# B&R Automation Studio project TD52 (part 62)

```c
  /* End of Outputs for SubSystem: '<S306>/2nd Order Filter1' */

  /* Outputs for Atomic SubSystem: '<S306>/2nd Order Filter2' */
  Gen2_ref_undOrderFilter(rtb_p2HP,
    Gen2_ref_B->BusInput3.fdc.r2ndOrdFiltOmegaPressure,
    Gen2_ref_B->BusInput3.fdc.r2ndOrdFiltDPressure, rtb_bResetBdc,
    &Gen2_ref_B->undOrderFilter2, &Gen2_ref_DWork->undOrderFilter2, inst);

  /* End of Outputs for SubSystem: '<S306>/2nd Order Filter2' */

  /* Outputs for Atomic SubSystem: '<S306>/2nd Order Filter3' */
  Gen2_ref_undOrderFilter3(rtb_p2s,
    Gen2_ref_B->BusInput3.fdc.r2ndOrdFiltOmegaPressure,
    Gen2_ref_B->BusInput3.fdc.r2ndOrdFiltDPressure, rtb_bResetBdc,
    &Gen2_ref_B->undOrderFilter3, &Gen2_ref_DWork->undOrderFilter3, inst);

  /* End of Outputs for SubSystem: '<S306>/2nd Order Filter3' */

  /* Switch: '<S272>/Switch2' */
  if (Gen2_ref_B->BusInput3.fdc.bEnable2ndOrdFiltDerivative) {
    /* Switch: '<S272>/Switch6' incorporates:
     *  Constant: '<S307>/Constant2'
     *  DiscreteIntegrator: '<S307>/Discrete-Time Integrator'
     *  Product: '<S307>/Product'
     *  Product: '<S307>/Product1'
     *  Sum: '<S307>/Sum'
     *  Sum: '<S307>/Sum4'
     */
    if (Gen2_ref_B->BusInput3.fdc.bEnableTransSwFilt) {
      rtb_Switch2_gd_idx_0 = (1.0 -
        Gen2_ref_DWork->DiscreteTimeIntegrator_DSTATE_d) *
        Gen2_ref_B->sf_FILTERnodelay.d_dt +
        Gen2_ref_DWork->DiscreteTimeIntegrator_DSTATE_d *
        Gen2_ref_B->undOrderFilter.Switch1;
      rtb_Switch2_gd_idx_1 = (1.0 -
        Gen2_ref_DWork->DiscreteTimeIntegrator_DSTATE_d) *
        Gen2_ref_B->sf_FILTERnodelay1.d_dt +
        Gen2_ref_DWork->DiscreteTimeIntegrator_DSTATE_d *
        Gen2_ref_B->undOrderFilter1.Switch1;
      rtb_Switch2_gd_idx_2 = (1.0 -
        Gen2_ref_DWork->DiscreteTimeIntegrator_DSTATE_d) *
        Gen2_ref_B->sf_FILTERnodelay2.d_dt +
        Gen2_ref_DWork->DiscreteTimeIntegrator_DSTATE_d *
        Gen2_ref_B->undOrderFilter2.Switch1;
      rtb_Switch2_gd_idx_3 = (1.0 -
        Gen2_ref_DWork->DiscreteTimeIntegrator_DSTATE_d) *
        Gen2_ref_B->sf_FILTERnodelay3.d_dt +
        Gen2_ref_DWork->DiscreteTimeIntegrator_DSTATE_d *
        Gen2_ref_B->undOrderFilter3.Switch1;
    } else {
      rtb_Switch2_gd_idx_0 = Gen2_ref_B->undOrderFilter.Switch1;
      rtb_Switch2_gd_idx_1 = Gen2_ref_B->undOrderFilter1.Switch1;
      rtb_Switch2_gd_idx_2 = Gen2_ref_B->undOrderFilter2.Switch1;
      rtb_Switch2_gd_idx_3 = Gen2_ref_B->undOrderFilter3.Switch1;
    }

    /* End of Switch: '<S272>/Switch6' */
  } else {
    rtb_Switch2_gd_idx_0 = Gen2_ref_B->sf_FILTERnodelay.d_dt;
    rtb_Switch2_gd_idx_1 = Gen2_ref_B->sf_FILTERnodelay1.d_dt;
    rtb_Switch2_gd_idx_2 = Gen2_ref_B->sf_FILTERnodelay2.d_dt;
    rtb_Switch2_gd_idx_3 = Gen2_ref_B->sf_FILTERnodelay3.d_dt;
  }

  /* End of Switch: '<S272>/Switch2' */

  /* DataTypeConversion: '<S4>/Data Type Conversion1' */
  rtb_Product1_b = Gen2_ref_B->BusInput.tT.rT1LP;

  /* Outputs for Atomic SubSystem: '<S196>/T1LP_filt' */
  /* Bias: '<S4>/C2K' */
  Gen2_ref_N_TC_HP_filt(rtb_Product1_b + 273.15,
                        Gen2_ref_B->BusInput3.inFilt.rTiF_T, rtb_bResetBdc,
                        &Gen2_ref_B->T1LP_filt, &Gen2_ref_DWork->T1LP_filt, inst);

  /* End of Outputs for SubSystem: '<S196>/T1LP_filt' */

  /* DataTypeConversion: '<S4>/Data Type Conversion8' */
  rtb_Product1_b = Gen2_ref_B->BusInput.tT.rT1HP;

  /* Outputs for Atomic SubSystem: '<S195>/T1HP_filt' */
  /* Bias: '<S4>/C2K1' */
  Gen2_ref_N_TC_HP_filt(rtb_Product1_b + 273.15,
                        Gen2_ref_B->BusInput3.inFilt.rTiF_T, rtb_bResetBdc,
                        &Gen2_ref_B->T1HP_filt, &Gen2_ref_DWork->T1HP_filt, inst);

  /* End of Outputs for SubSystem: '<S195>/T1HP_filt' */

  /* Outputs for Atomic SubSystem: '<S267>/Mg' */
  Gen2_ref_Mg(Gen2_ref_B->BusInput3.eng.rRho_gas, &Gen2_ref_B->Mg, inst);

  /* End of Outputs for SubSystem: '<S267>/Mg' */

  /* Sum: '<S342>/Sum2' */
  rtb_Switch1_k = u0;

  /* Abs: '<S342>/Abs3' */
  rtb_Switch_jv = fabs(rtb_Switch1_k);

  /* Sum: '<S381>/Add1' */
  rtb_Product1_b = Gen2_ref_B->BusInput3.EGTLim.rT_CR_soft -
    Gen2_ref_B->BusInput3.EGTLim.rT_CR_hard;

  /* Saturate: '<S381>/Saturation6' */
  if (rtb_Product1_b > 1.0E+6) {
    rtb_Saturation6 = 1.0E+6;
  } else if (rtb_Product1_b < 1.0) {
    rtb_Saturation6 = 1.0;
  } else {
    rtb_Saturation6 = rtb_Product1_b;
  }

  /* End of Saturate: '<S381>/Saturation6' */

  /* DataTypeConversion: '<S4>/Data Type Conversion12' */
  rtb_Product1_b = Gen2_ref_B->BusInput.tT.rTcylMax;

  /* Bias: '<S342>/Bias' incorporates:
   *  Bias: '<S4>/C2K5'
   */
  rtb_PactOut_o = (rtb_Product1_b + 273.15) + -273.15;

  /* Sum: '<S381>/Add6' */
  rtb_Divide6_n = Gen2_ref_B->BusInput3.EGTLim.rT_max -
    Gen2_ref_B->BusInput3.EGTLim.rT_CR_hard;

  /* Sum: '<S381>/Sum15' */
  rtb_Switch2_n5 = (rtb_PactOut_o + rtb_Saturation6) - rtb_Divide6_n;

  /* Switch: '<S387>/Switch2' incorporates:
   *  Constant: '<S381>/Constant17'
   *  RelationalOperator: '<S387>/LowerRelop1'
   *  RelationalOperator: '<S387>/UpperRelop'
   *  Switch: '<S387>/Switch'
   */
  if (rtb_Switch2_n5 > rtb_Saturation6) {
    rtb_Switch2_n5 = rtb_Saturation6;
  } else if (rtb_Switch2_n5 < 0.0) {
    /* Switch: '<S387>/Switch' incorporates:
     *  Constant: '<S381>/Constant17'
     */
    rtb_Switch2_n5 = 0.0;
  }

  /* End of Switch: '<S387>/Switch2' */

  /* Switch: '<S381>/Switch7' incorporates:
   *  Constant: '<S381>/Constant23'
   *  Constant: '<S381>/Constant5'
   *  Product: '<S381>/Divide8'
   *  Sum: '<S381>/Sum1'
   */
  if (Gen2_ref_B->BusInput3.EGTLim.bActive) {
    rtb_Product1_b = 1.0 - rtb_Switch2_n5 / rtb_Saturation6;
  } else {
    rtb_Product1_b = 1.0;
  }

  /* End of Switch: '<S381>/Switch7' */

  /* Product: '<S342>/Product' */
  rtb_Product1_b *= rtb_Switch_jv;

  /* Switch: '<S380>/Switch2' incorporates:
   *  RelationalOperator: '<S380>/LowerRelop1'
   */
  if (!(rtb_Switch1_k > rtb_Product1_b)) {
    /* Gain: '<S342>/Gain2' */
    rtb_Switch_jv = -rtb_Switch_jv;

    /* Switch: '<S380>/Switch' incorporates:
     *  RelationalOperator: '<S380>/UpperRelop'
     */
    if (rtb_Switch1_k < rtb_Switch_jv) {
      rtb_Product1_b = rtb_Switch_jv;
    } else {
      rtb_Product1_b = rtb_Switch1_k;
    }

    /* End of Switch: '<S380>/Switch' */
  }

  /* End of Switch: '<S380>/Switch2' */

  /* Gain: '<S342>/Gain4' */
  rtb_Switch_jv = -1.0E-6 * rtb_Product1_b;

  /* Sum: '<S11>/Sum' incorporates:
   *  Constant: '<S11>/Constant'
   */
  rtb_Switch_fy_tmp_tmp = 1.0 - Gen2_ref_B->BusInput.IN_EC_rGT_RatioMix_TC2;
  rtb_Product1_b = 1.0 - Gen2_ref_B->BusInput.IN_EC_rGT_RatioMix_TC2;

  /* Saturate: '<S11>/Saturation' */
  if (rtb_Product1_b > 1.0) {
    rtb_Product1_b = 1.0;
  } else if (rtb_Product1_b < 0.0) {
    rtb_Product1_b = 0.0;
  }

  /* End of Saturate: '<S11>/Saturation' */

  /* Saturate: '<S11>/Saturation1' */
  if (Gen2_ref_B->BusInput.IN_EC_rGT_RatioMix_TC2 > 1.0F) {
    rtb_rPos_CBV3 = 1.0F;
  } else if (Gen2_ref_B->BusInput.IN_EC_rGT_RatioMix_TC2 < 0.0F) {
    rtb_rPos_CBV3 = 0.0F;
  } else {
    rtb_rPos_CBV3 = Gen2_ref_B->BusInput.IN_EC_rGT_RatioMix_TC2;
  }

  /* End of Saturate: '<S11>/Saturation1' */

  /* Sum: '<S11>/Sum1' incorporates:
   *  Product: '<S11>/Product'
   *  Product: '<S11>/Product1'
   */
  rtb_Sum1_idx_2 = rtb_Product1_b * Gen2_ref_B->BusInput3.eng.rMin_Air_Ratio_kg
    + rtb_rPos_CBV3 * Gen2_ref_B->BusInput3.eng.rMin_Air_Ratio_M_kg;
  rtb_Sum1_idx_3 = rtb_Product1_b * Gen2_ref_B->BusInput3.eng.rLHV +
    rtb_rPos_CBV3 * Gen2_ref_B->BusInput3.eng.rLHV_M;

  /* Switch: '<S3>/etaVolConst' */
  if (Gen2_ref_B->BusInput3.Eff.bActive_EtaVolExt) {
    rtb_etaVolConst_lt = Gen2_ref_B->BusInput3.Eff.rEtaVolExt;
  } else {
    rtb_etaVolConst_lt = 0.0;
  }

  /* End of Switch: '<S3>/etaVolConst' */

  /* Switch: '<S3>/etaBreakConst' */
  if (Gen2_ref_B->BusInput3.Eff.bActive_EtaBrakeExt) {
    rtb_etaBreakConst = Gen2_ref_B->BusInput3.Eff.rEtaBrakeExt;
  } else {
    rtb_etaBreakConst = 0.0;
  }

  /* End of Switch: '<S3>/etaBreakConst' */

  /* Switch: '<S342>/Switch' */
  if (Gen2_ref_B->BusInput3.PowCtrl.bActive_MbcFF) {
    /* Product: '<S340>/Divide1' incorporates:
     *  Constant: '<S340>/Constant'
     *  Constant: '<S340>/R_air'
     */
    rtb_Switch1_k = rtb_Sum1_idx_2 * 287.15 * Gen2_ref_B->T2s_filt.Switch *
      rtb_kW2W1_h * 12.566370614359172;

    /* Saturate: '<S340>/Saturation1' */
    if (rtb_Switch1_k <= 1.0) {
      rtb_Switch1_k = 1.0;
    }

    /* End of Saturate: '<S340>/Saturation1' */

    /* Saturate: '<S340>/Saturation' */
    if (rtb_Sum1_idx_2 <= 1.0) {
      rtb_Product1_b = 1.0;
    } else {
      rtb_Product1_b = rtb_Sum1_idx_2;
    }

    /* End of Saturate: '<S340>/Saturation' */

    /* Sum: '<S340>/Sum' incorporates:
     *  Constant: '<S340>/Constant1'
     *  Gain: '<S340>/Gain'
     *  Product: '<S340>/Divide'
     *  Product: '<S340>/Divide2'
     *  Product: '<S340>/Divide4'
     */
    rtb_Switch_e3 = Gen2_ref_B->BusInput3.eng.rVol_Hub_Eng * rtb_Sum1_idx_3 *
      (0.10471975511965977 * Gen2_ref_B->BusInput3.eng.rN_Nom) *
      rtb_etaVolConst_lt * rtb_etaBreakConst * Gen2_ref_B->p2s_filt.Switch /
      rtb_Switch1_k - 1.0 / rtb_Product1_b;

    /* Saturate: '<S340>/Saturation2' */
    if (rtb_Switch_e3 > 2.2) {
      rtb_Switch_e3 = 2.2;
    } else if (rtb_Switch_e3 < 1.3) {
      rtb_Switch_e3 = 1.3;
    }

    /* End of Saturate: '<S340>/Saturation2' */
  } else {
    rtb_Switch_e3 = Gen2_ref_B->BusInput3.PowCtrl.rLam_ff;
  }

  /* End of Switch: '<S342>/Switch' */

  /* Switch: '<S381>/Switch8' incorporates:
   *  Constant: '<S381>/Constant10'
   *  Product: '<S381>/Product'
   *  Product: '<S381>/Product1'
   *  Sum: '<S381>/Sum16'
   */
  if (Gen2_ref_B->BusInput3.EGTLim.bActive) {
    /* Sum: '<S381>/Sum8' */
    u0 = rtb_PactOut_o - rtb_Divide6_n;

    /* Saturate: '<S381>/Saturation3' */
    if (u0 > 1.0E+6) {
      u0 = 1.0E+6;
    } else if (u0 < 0.0) {
      u0 = 0.0;
    }

    /* End of Saturate: '<S381>/Saturation3' */
    rtb_Switch8 = u0 * Gen2_ref_B->BusInput3.EGTLim.rKaw_hard +
      Gen2_ref_B->BusInput3.EGTLim.rKaw_soft * rtb_Switch2_n5;
  } else {
    rtb_Switch8 = 0.0;
  }

  /* End of Switch: '<S381>/Switch8' */

  /* Gain: '<S14>/Gain2' incorporates:
   *  Gain: '<S133>/Gain1'
   *  Gain: '<S14>/Gain'
   *  Gain: '<S14>/Gain3'
   *  Gain: '<S23>/Gain'
   *  Gain: '<S25>/Gain1'
   *  Gain: '<S426>/Gain1'
   *  Gain: '<S9>/Gain5'
   *  Switch: '<S106>/Switch2'
   *  Switch: '<S133>/Switch'
   *  Switch: '<S133>/Switch1'
   *  Switch: '<S426>/Switch'
   *  Switch: '<S426>/Switch1'
   *  Switch: '<S426>/Switch2'
   *  Switch: '<S494>/etaVolConst'
   */
  rtb_kW2W1_h = 1.0E-5 * Gen2_ref_B->p2s_filt.Switch;
  rtb_Product1_b = rtb_kW2W1_h;

  /* S-Function (sfix_look1_dyn): '<S14>/Lookup Table Dynamic1' */
  /* Dynamic Look-Up Table Block: '<S14>/Lookup Table Dynamic1'
   * Input0  Data Type:  Floating Point real_T
   * Input1  Data Type:  Floating Point real_T
   * Input2  Data Type:  Floating Point real_T
   * Output0 Data Type:  Floating Point real_T
   * Saturation Mode: Saturate
   * Lookup Method: Linear_Endpoint
   *
   */
  LookUp_real_T_real_T_SAT( &(rtb_Sum8_m),
    &Gen2_ref_B->BusInput3.LamLim.refPoint_LamUpLim_ABS_y[0], rtb_Product1_b,
    &Gen2_ref_B->BusInput3.LamLim.refPoint_LamUpLim_ABS_x[0], 5U, inst);

  /* Logic: '<S14>/Logical Operator6' incorporates:
   *  Logic: '<S14>/Logical Operator10'
   */
  rtb_LogicalOperator5_g_tmp =
    !Gen2_ref_B->BusInput3.LamLim.bActLamLim_GQCimprovement;

  /* Logic: '<S14>/Logical Operator5' incorporates:
   *  Logic: '<S14>/Logical Operator6'
   */
  rtb_LogicalOperator5_mv = (Gen2_ref_B->BusInput3.LamLim.bLamOffsInitPerm ||
    rtb_LogicalOperator5_g_tmp);

  /* Gain: '<S14>/Gain3' */
  rtb_Product1_b = rtb_kW2W1_h;

  /* S-Function (sfix_look1_dyn): '<S14>/Lookup Table Dynamic2' */
  /* Dynamic Look-Up Table Block: '<S14>/Lookup Table Dynamic2'
   * Input0  Data Type:  Floating Point real_T
   * Input1  Data Type:  Floating Point real_T
   * Input2  Data Type:  Floating Point real_T
   * Output0 Data Type:  Floating Point real_T
   * Saturation Mode: Saturate
   * Lookup Method: Linear_Endpoint
   *
   */
  LookUp_real_T_real_T_SAT( &(rtb_LookupTableDynamic2),
    &Gen2_ref_B->BusInput3.LamLim.refPoint_LamLoLim_ABS_y[0], rtb_Product1_b,
    &Gen2_ref_B->BusInput3.LamLim.refPoint_LamLoLim_ABS_x[0], 5U, inst);

  /* Saturate: '<S14>/Saturation' */
  if (Gen2_ref_B->BusInput3.LamLim.rFactEnrich <= 0.0) {
    rtb_Product1_b = 0.0;
  } else {
    rtb_Product1_b = Gen2_ref_B->BusInput3.LamLim.rFactEnrich;
  }

  /* End of Saturate: '<S14>/Saturation' */

  /* Gain: '<S14>/Gain' */
  rtb_PactOut_o = rtb_kW2W1_h;

  /* Switch: '<S14>/Switch5' */
  if (Gen2_ref_B->BusInput3.LamLim.bNOx250mg) {
    /* S-Function (sfix_look1_dyn): '<S14>/Lookup Table Dynamic' */
    /* Dynamic Look-Up Table Block: '<S14>/Lookup Table Dynamic'
     * Input0  Data Type:  Floating Point real_T
     * Input1  Data Type:  Floating Point real_T
     * Input2  Data Type:  Floating Point real32_T
     * Output0 Data Type:  Floating Point real_T
     * Saturation Mode: Saturate
     * Lookup Method: Linear_Endpoint
     *
     */
    LookUp_real_Treal32_T_K4km1JJi( &(rtb_LookupTableDynamic_n),
      &Gen2_ref_B->BusInput3.LamLim.rLamMapBase250mg[0], rtb_PactOut_o,
      &Gen2_ref_B->BusInput3.LamLim.rPr_p2s_Lup_in[0], 9U, inst);
    rtb_PactOut_o = rtb_LookupTableDynamic_n;
  } else {
    /* S-Function (sfix_look1_dyn): '<S14>/Lookup Table Dynamic3' */
    /* Dynamic Look-Up Table Block: '<S14>/Lookup Table Dynamic3'
     * Input0  Data Type:  Floating Point real_T
     * Input1  Data Type:  Floating Point real_T
     * Input2  Data Type:  Floating Point real32_T
     * Output0 Data Type:  Floating Point real_T
     * Saturation Mode: Saturate
     * Lookup Method: Linear_Endpoint
     *
     */
    LookUp_real_Treal32_T_K4km1JJi( &(rtb_LookupTableDynamic3),
      &Gen2_ref_B->BusInput3.LamLim.rLamMapBase[0], rtb_PactOut_o,
      &Gen2_ref_B->BusInput3.LamLim.rPr_p2s_Lup_in[0], 9U, inst);
    rtb_PactOut_o = rtb_LookupTableDynamic3;
  }

  /* End of Switch: '<S14>/Switch5' */

  /* Product: '<S14>/Product' incorporates:
   *  Constant: '<S14>/Constant'
   *  Sum: '<S14>/Sum1'
   *  Sum: '<S14>/Sum2'
   */
  rtb_Product_l0 = (1.0 - rtb_Product1_b) * (rtb_PactOut_o -
    rtb_LookupTableDynamic2);

  /* Delay: '<S14>/Resettable Delay2' */
  if (Gen2_ref_DWork->icLoad_l) {
    Gen2_ref_DWork->ResettableDelay2_DSTATE =
      Gen2_ref_B->BusInput3.LamLim.rLamOffsetLimInit;
  }

  rtb_Product1_b = Gen2_ref_DWork->ResettableDelay2_DSTATE;

  /* End of Delay: '<S14>/Resettable Delay2' */

  /* Switch: '<S14>/Switch6' incorporates:
   *  DataTypeConversion: '<S4>/Data Type Conversion28'
   *  DataTypeConversion: '<S4>/Data Type Conversion31'
   *  DataTypeConversion: '<S4>/Data Type Conversion32'
   *  Sum: '<S14>/Sum16'
   *  UnitDelay: '<S14>/Unit Delay4'
   */
  if (Gen2_ref_DWork->UnitDelay4_DSTATE_d) {
    rtb_Divide6_n = (((Gen2_ref_B->BusInput.rLam_idle - rtb_LookupTableDynamic2)
                      - rtb_Product_l0) - Gen2_ref_B->BusInput.rOffsetLamLimit)
      + Gen2_ref_B->BusInput.rDeltaLamSync;
  } else {
    rtb_Divide6_n = rtb_Product1_b;
  }

  /* End of Switch: '<S14>/Switch6' */

  /* Switch: '<S14>/Switch7' */
  if (rtb_LogicalOperator5_mv) {
    rtb_Switch2_n5 = Gen2_ref_B->BusInput3.LamLim.rLamOffsetLimInit;
  } else {
    rtb_Switch2_n5 = rtb_Divide6_n;
  }

  /* End of Switch: '<S14>/Switch7' */

  /* Delay: '<S14>/Resettable Delay' incorporates:
   *  Logic: '<Root>/Logical Operator'
   */
  Gen2_ref_DWork->icLoad_i =
    ((((Gen2_ref_PrevZCSigState->ResettableDelay_Reset_ZCE_j == 1) != (int32_T)
       rtb_LogicalOperator_cn) &&
      (Gen2_ref_PrevZCSigState->ResettableDelay_Reset_ZCE_j != 3)) ||
     rtb_LogicalOperator_cn || Gen2_ref_DWork->icLoad_i);
  Gen2_ref_PrevZCSigState->ResettableDelay_Reset_ZCE_j = rtb_LogicalOperator_cn;
  if (Gen2_ref_DWork->icLoad_i) {
    Gen2_ref_DWork->ResettableDelay_DSTATE_l = rtb_Switch2_n5;
  }

  /* Sum: '<S14>/Sum' incorporates:
   *  DataTypeConversion: '<S4>/Data Type Conversion28'
   *  UnitDelay: '<S14>/Unit Delay'
   */
  rtb_Switch1_k = (Gen2_ref_DWork->UnitDelay_DSTATE -
                   Gen2_ref_B->BusInput.rOffsetLamLimit) - rtb_PactOut_o;

  /* Switch: '<S14>/Switch9' */
  if (rtb_Switch2_jv) {
    /* Switch: '<S860>/Switch2' incorporates:
     *  Constant: '<S14>/Constant2'
     *  Delay: '<S14>/Resettable Delay'
     *  RelationalOperator: '<S860>/LowerRelop1'
     *  RelationalOperator: '<S860>/UpperRelop'
     *  Switch: '<S860>/Switch'
     */
    if (rtb_Switch1_k > 2.0) {
      rtb_Switch1_k = 2.0;
    } else if (rtb_Switch1_k < Gen2_ref_DWork->ResettableDelay_DSTATE_l) {
      /* Switch: '<S860>/Switch' incorporates:
       *  Delay: '<S14>/Resettable Delay'
       */
      rtb_Switch1_k = Gen2_ref_DWork->ResettableDelay_DSTATE_l;
    }

    /* End of Switch: '<S860>/Switch2' */
  }

  /* End of Switch: '<S14>/Switch9' */

  /* Abs: '<S858>/Abs' */
  rtb_Product1_b = rtb_Product1_e_tmp;

  /* Switch: '<S858>/Switch' incorporates:
   *  Constant: '<S858>/Constant2'
   *  RelationalOperator: '<S858>/Relational Operator'
   */
  if (2.2204460492503131E-16 >= rtb_Product1_b) {
    rtb_bResetHlci_0 = 2.2204460492503131E-16;
  } else {
    rtb_bResetHlci_0 = Gen2_ref_B->BusInput3.eng.rP_Nom;
  }

  /* End of Switch: '<S858>/Switch' */

  /* RelationalOperator: '<S14>/Relational Operator' incorporates:
   *  Gain: '<S14>/Gain1'
   *  Product: '<S14>/Divide'
   */
  rtb_RelationalOperator_l5 = (0.001 * rtb_Gain2_ao / rtb_bResetHlci_0 >
    Gen2_ref_B->BusInput3.LamLim.rPminSSadapt);

  /* Switch: '<S908>/Switch' incorporates:
   *  Constant: '<S908>/Constant2'
   *  RelationalOperator: '<S908>/Relational Operator'
   */
  if (2.2204460492503131E-16 >= rtb_Product1_b) {
    rtb_bResetHlci_0 = 2.2204460492503131E-16;
  } else {
    rtb_bResetHlci_0 = Gen2_ref_B->BusInput3.eng.rP_Nom;
  }

  /* End of Switch: '<S908>/Switch' */

  /* Product: '<S20>/Divide1' incorporates:
   *  Gain: '<S20>/Gain6'
   */
  rtb_Saturation6 = 0.001 * rtb_Gain2_ao / rtb_bResetHlci_0;

  /* Outputs for Atomic SubSystem: '<S20>/Filter1' */
  /* Logic: '<Root>/Logical Operator' */
  Gen2_ref_Filter3(rtb_Saturation6, Gen2_ref_B->BusInput3.LamLim.rTiSSfilter,
                   Gen2_ref_ConstB.T_filt1, rtb_LogicalOperator_cn,
                   &Gen2_ref_B->Filter1_ny, &Gen2_ref_DWork->Filter1_ny, inst);

  /* End of Outputs for SubSystem: '<S20>/Filter1' */

  /* Logic: '<S917>/Logical Operator' incorporates:
   *  Logic: '<Root>/Logical Operator'
   *  UnitDelay: '<S917>/Unit Delay'
   */
  rtb_LogicalOperator_i = (rtb_LogicalOperator_cn ||
    Gen2_ref_DWork->UnitDelay_DSTATE_k);

  /* DiscreteIntegrator: '<S917>/Discrete-Time Integrator' */
  if (rtb_LogicalOperator_i || (Gen2_ref_DWork->DiscreteTimeIntegrator_PrevR_ka
       != 0)) {
    Gen2_ref_DWork->DiscreteTimeIntegrator_DSTATE_c = 0.0;
  }

  /* RelationalOperator: '<S917>/Relational Operator' incorporates:
   *  DiscreteIntegrator: '<S917>/Discrete-Time Integrator'
   */
  rtb_RelationalOperator_a = (Gen2_ref_B->BusInput3.LamLim.rTiSSsampling <=
    Gen2_ref_DWork->DiscreteTimeIntegrator_DSTATE_c);

  /* Outputs for Enabled SubSystem: '<S20>/Enabled Subsystem2' incorporates:
   *  EnablePort: '<S909>/Enable'
   */
  if (rtb_RelationalOperator_a) {
    /* Inport: '<S909>/In1' */
    Gen2_ref_B->In1 = Gen2_ref_B->Filter1_ny.Switch;

    /* Memory: '<S909>/Memory' */
    FILT_IN = Gen2_ref_DWork->Memory_PreviousInput;

    /* Sum: '<S909>/Sum' */
    Gen2_ref_B->Sum = Gen2_ref_B->In1 - FILT_IN;

    /* Update for Memory: '<S909>/Memory' */
    Gen2_ref_DWork->Memory_PreviousInput = Gen2_ref_B->In1;
  }

  /* End of Outputs for SubSystem: '<S20>/Enabled Subsystem2' */

  /* Sum: '<S20>/Sum2' */
  rtb_Product1_b = rtb_Saturation6 - Gen2_ref_B->In1;

  /* Abs: '<S20>/Abs4' */
  rtb_Saturation6 = fabs(rtb_Product1_b);

  /* Outputs for Atomic SubSystem: '<S20>/Filter3' */
  /* Logic: '<Root>/Logical Operator' */
  Gen2_ref_Filter3(rtb_Saturation6, Gen2_ref_B->BusInput3.LamLim.rTiSSfilter,
                   Gen2_ref_ConstB.T_filt1, rtb_LogicalOperator_cn,
                   &Gen2_ref_B->Filter3_f, &Gen2_ref_DWork->Filter3_f, inst);

  /* End of Outputs for SubSystem: '<S20>/Filter3' */

  /* Abs: '<S20>/Abs1' */
  rtb_Product1_b = fabs(Gen2_ref_B->Sum);

  /* RelationalOperator: '<S20>/Relational Operator3' */
  rtb_LogicalOperator_aw = (rtb_Product1_b <=
    Gen2_ref_B->BusInput3.LamLim.rThrshSSPow);

  /* Gain: '<S20>/Gain1' incorporates:
   *  Sum: '<S20>/Sum'
   */
  rtb_Product1_b = (Gen2_ref_B->p2s_filt.Switch - rtb_Divide_kt) * 0.01;

  /* Abs: '<S20>/Abs' */
  rtb_Abs = fabs(rtb_Product1_b);

  /* Gain: '<S20>/Gain2' */
  rtb_Product1_b = 2.0 * Gen2_ref_B->BusInput3.LamLim.rThrshSSboost;

  /* Outputs for Atomic SubSystem: '<S20>/Filter' */
  /* Logic: '<Root>/Logical Operator' */
  Gen2_ref_Filter3(rtb_Abs, Gen2_ref_B->BusInput3.LamLim.rTiSSfilter,
                   Gen2_ref_ConstB.T_filt1, rtb_LogicalOperator_cn,
                   &Gen2_ref_B->Filter_f, &Gen2_ref_DWork->Filter_f, inst);

  /* End of Outputs for SubSystem: '<S20>/Filter' */

  /* Outputs for Atomic SubSystem: '<S20>/TON1' */
  /* Logic: '<S20>/Logical Operator' incorporates:
   *  RelationalOperator: '<S20>/Relational Operator'
   *  RelationalOperator: '<S20>/Relational Operator1'
   */
  Gen2_ref_TON_1(((rtb_Abs <= rtb_Product1_b) && (Gen2_ref_B->Filter_f.Switch <=
    Gen2_ref_B->BusInput3.LamLim.rThrshSSboost)),
                 Gen2_ref_B->BusInput3.LamLim.rTiSSsampling, &Gen2_ref_B->TON1_n,
                 &Gen2_ref_DWork->TON1_n, inst);

  /* End of Outputs for SubSystem: '<S20>/TON1' */

  /* Sum: '<S20>/Sum1' incorporates:
   *  DataTypeConversion: '<S4>/Data Type Conversion16'
   */
  rtb_Product1_b = rtb_DataTypeConversion15 - Gen2_ref_B->BusInput.rN_Set;

  /* Abs: '<S20>/Abs3' */
  rtb_Abs = fabs(rtb_Product1_b);

  /* Gain: '<S20>/Gain3' */
  rtb_Product1_b = 2.0 * Gen2_ref_B->BusInput3.LamLim.rThrshSSspeed;

  /* Outputs for Atomic SubSystem: '<S20>/Filter2' */
  /* Logic: '<Root>/Logical Operator' */
  Gen2_ref_Filter3(rtb_Abs, Gen2_ref_B->BusInput3.LamLim.rTiSSfilter,
                   Gen2_ref_ConstB.T_filt1, rtb_LogicalOperator_cn,
                   &Gen2_ref_B->Filter2_o, &Gen2_ref_DWork->Filter2_o, inst);

  /* End of Outputs for SubSystem: '<S20>/Filter2' */

  /* Outputs for Atomic SubSystem: '<S20>/TON' */
  /* Logic: '<S20>/Logical Operator2' incorporates:
   *  RelationalOperator: '<S20>/Relational Operator4'
   *  RelationalOperator: '<S20>/Relational Operator5'
   */
  Gen2_ref_TON_1(((rtb_Abs <= rtb_Product1_b) && (Gen2_ref_B->Filter2_o.Switch <=
    Gen2_ref_B->BusInput3.LamLim.rThrshSSspeed)),
                 Gen2_ref_B->BusInput3.LamLim.rTiSSsampling, &Gen2_ref_B->TON_l,
                 &Gen2_ref_DWork->TON_l, inst);

  /* End of Outputs for SubSystem: '<S20>/TON' */

  /* Outputs for Atomic SubSystem: '<S20>/TON2' */
  /* Logic: '<S20>/Logical Operator1' incorporates:
   *  RelationalOperator: '<S20>/Relational Operator2'
   *  RelationalOperator: '<S20>/Relational Operator6'
   */
  Gen2_ref_TON_1(((rtb_Saturation6 <= Gen2_ref_B->BusInput3.LamLim.rThrshSSPow) &&
                  (Gen2_ref_B->Filter3_f.Switch <=
                   Gen2_ref_B->BusInput3.LamLim.rThrshSSPow) &&
                  rtb_LogicalOperator_aw && Gen2_ref_B->TON1_n.LogicalOperator3 &&
                  Gen2_ref_B->TON_l.LogicalOperator3),
                 Gen2_ref_B->BusInput3.LamLim.rTiSSsampling, &Gen2_ref_B->TON2,
                 &Gen2_ref_DWork->TON2, inst);

  /* End of Outputs for SubSystem: '<S20>/TON2' */

  /* Switch: '<S14>/Switch4' incorporates:
   *  Delay: '<S14>/Resettable Delay'
   *  Logic: '<S14>/Logical Operator1'
   *  Switch: '<S14>/Switch3'
   */
  if (rtb_RelationalOperator_l5 &&
      Gen2_ref_B->BusInput3.LamLim.bAutomaticOffsetON &&
      (Gen2_ref_B->BusInput3.LamLim.bActLambdaOffsetNotSteady ||
       Gen2_ref_B->TON2.LogicalOperator3)) {
    /* Switch: '<S14>/Switch12' */
    if (rtb_Switch4_mu) {
      /* Switch: '<S861>/Switch2' incorporates:
       *  Constant: '<S14>/Constant6'
       *  Delay: '<S14>/Resettable Delay'
       *  RelationalOperator: '<S861>/LowerRelop1'
       *  RelationalOperator: '<S861>/UpperRelop'
       *  Switch: '<S861>/Switch'
       */
      if (rtb_Switch1_k > Gen2_ref_DWork->ResettableDelay_DSTATE_l) {
        rtb_Switch1_k = Gen2_ref_DWork->ResettableDelay_DSTATE_l;
      } else if (rtb_Switch1_k < -2.0) {
        /* Switch: '<S861>/Switch' incorporates:
         *  Constant: '<S14>/Constant6'
         */
        rtb_Switch1_k = -2.0;
      }

      /* End of Switch: '<S861>/Switch2' */
    }

    /* End of Switch: '<S14>/Switch12' */
  } else {
    rtb_Switch1_k = Gen2_ref_DWork->ResettableDelay_DSTATE_l;
  }

  /* End of Switch: '<S14>/Switch4' */

  /* Switch: '<S14>/Switch10' incorporates:
   *  Logic: '<S14>/Logical Operator7'
   *  Logic: '<S14>/Logical Operator9'
   *  Product: '<S14>/Divide1'
   */
  if (Gen2_ref_B->TON2.LogicalOperator3 ||
      (!Gen2_ref_B->BusInput3.LamLim.bActLambdaOffsetNotSteady)) {
    rtb_bResetHlci_0 = Gen2_ref_B->BusInput3.LamLim.rTiFiltLambdaOffset;
  } else {
    rtb_bResetHlci_0 = Gen2_ref_B->BusInput3.LamLim.rFactTiFiltLamOffsNotSteady *
      Gen2_ref_B->BusInput3.LamLim.rTiFiltLambdaOffset;
  }

  /* End of Switch: '<S14>/Switch10' */

  /* Outputs for Atomic SubSystem: '<S14>/Filter' */
  /* Logic: '<Root>/Logical Operator' */
  Gen2_ref_Pd_filt(rtb_Switch1_k, rtb_bResetHlci_0, rtb_Switch2_n5,
                   rtb_LogicalOperator_cn, &Gen2_ref_B->Filter_l,
                   &Gen2_ref_DWork->Filter_l, inst);

  /* End of Outputs for SubSystem: '<S14>/Filter' */

  /* Sum: '<S14>/Sum4' incorporates:
   *  DataTypeConversion: '<S4>/Data Type Conversion28'
   */
  rtb_Sum4_ny = Gen2_ref_B->Filter_l.Switch +
    Gen2_ref_B->BusInput.rOffsetLamLimit;

  /* Saturate: '<S14>/Saturation1' */
  if (Gen2_ref_B->BusInput3.LamLim.rFactLean <= 0.0) {
    rtb_Product1_b = 0.0;
  } else {
    rtb_Product1_b = Gen2_ref_B->BusInput3.LamLim.rFactLean;
  }

  /* End of Saturate: '<S14>/Saturation1' */

  /* Product: '<S14>/Product1' incorporates:
   *  Constant: '<S14>/Constant1'
   *  Sum: '<S14>/Sum6'
   *  Sum: '<S14>/Sum7'
   */
  rtb_Product1_b = (rtb_PactOut_o - rtb_Sum8_m) * (1.0 - rtb_Product1_b);

  /* Sum: '<S14>/Sum5' */
  rtb_Sum5_j = rtb_Sum4_ny + rtb_Product1_b;

  /* Sum: '<S14>/Sum3' */
  rtb_Switch2_n5 = rtb_Sum8_m + rtb_Sum5_j;

  /* MinMax: '<S14>/MinMax' */
  if ((!(rtb_Switch2_n5 <= Gen2_ref_B->BusInput3.LamLim.rLam_max)) && (!rtIsNaN
       (Gen2_ref_B->BusInput3.LamLim.rLam_max))) {
    rtb_Switch2_n5 = Gen2_ref_B->BusInput3.LamLim.rLam_max;
  }

  /* End of MinMax: '<S14>/MinMax' */

  /* Sum: '<S14>/Sum8' */
  rtb_Sum8_m = rtb_Sum4_ny + rtb_Product_l0;

  /* Delay: '<S14>/Resettable Delay3' incorporates:
   *  Logic: '<Root>/Logical Operator'
   */
  Gen2_ref_DWork->icLoad_f =
    ((((Gen2_ref_PrevZCSigState->ResettableDelay3_Reset_ZCE == 1) != (int32_T)
       rtb_LogicalOperator_cn) &&
      (Gen2_ref_PrevZCSigState->ResettableDelay3_Reset_ZCE != 3)) ||
     rtb_LogicalOperator_cn || Gen2_ref_DWork->icLoad_f);
  Gen2_ref_PrevZCSigState->ResettableDelay3_Reset_ZCE = rtb_LogicalOperator_cn;
  Gen2_ref_DWork->ResettableDelay3_DSTATE = (Gen2_ref_DWork->icLoad_f ||
    Gen2_ref_DWork->ResettableDelay3_DSTATE);

  /* Switch: '<S14>/Switch13' incorporates:
   *  Constant: '<S14>/Constant5'
   *  Delay: '<S14>/Resettable Delay3'
   *  Logic: '<S14>/Logical Operator11'
   */
  if (Gen2_ref_DWork->ResettableDelay3_DSTATE) {
    rtb_RelationalOperator_l5 = !rtb_RelationalOperator_l5;
  } else {
    rtb_RelationalOperator_l5 = false;
  }

  /* End of Switch: '<S14>/Switch13' */

  /* Logic: '<S14>/Logical Operator12' */
  rtb_LogicalOperator12_a = !rtb_RelationalOperator_l5;

  /* Switch: '<S14>/Switch11' incorporates:
   *  Logic: '<Root>/Logical Operator'
   *  Logic: '<S14>/Logical Operator4'
   */
  if (rtb_LogicalOperator_cn || rtb_LogicalOperator12_a ||
      rtb_LogicalOperator5_g_tmp) {
    /* Sum: '<S14>/Sum9' */
    rtb_Switch1_k = rtb_LookupTableDynamic2 + rtb_Sum8_m;

    /* MinMax: '<S14>/MinMax1' */
    if ((!(rtb_Switch1_k >= Gen2_ref_B->BusInput3.LamLim.rLam_min)) && (!rtIsNaN
         (Gen2_ref_B->BusInput3.LamLim.rLam_min))) {
      rtb_Switch1_k = Gen2_ref_B->BusInput3.LamLim.rLam_min;
    }
  } else {
    /* Sum: '<S14>/Sum9' */
    u0 = rtb_LookupTableDynamic2 + rtb_Sum8_m;

    /* MinMax: '<S14>/MinMax1' */
    if ((!(u0 >= Gen2_ref_B->BusInput3.LamLim.rLam_min)) && (!rtIsNaN
         (Gen2_ref_B->BusInput3.LamLim.rLam_min))) {
      u0 = Gen2_ref_B->BusInput3.LamLim.rLam_min;
    }

    /* Sum: '<S14>/Sum14' incorporates:
     *  DataTypeConversion: '<S4>/Data Type Conversion31'
     *  DataTypeConversion: '<S4>/Data Type Conversion32'
     */
    rtb_Switch1_k = (real_T)Gen2_ref_B->BusInput.rLam_idle +
      Gen2_ref_B->BusInput.rDeltaLamSync;

    /* MinMax: '<S14>/MinMax4' */
    if ((u0 >= rtb_Switch1_k) || rtIsNaN(rtb_Switch1_k)) {
      rtb_Switch1_k = u0;
    }

    /* End of MinMax: '<S14>/MinMax4' */
  }

  /* End of Switch: '<S14>/Switch11' */

  /* Outputs for Atomic SubSystem: '<S342>/PID_Power' */
  /* Product: '<S379>/Divide1' */
  FILT_IN = Gen2_ref_B->BusInput3.PowCtrl.rKp * rtb_Switch_jv;

  /* BusCreator: '<Root>/Bus Creator' incorporates:
   *  BusCreator: '<S379>/Bus Creator1'
   *  DataTypeConversion: '<S379>/Data Type Conversion1'
   *  Outport: '<Root>/dbg'
   */
  Gen2_ref_Y->dbg.HLC.BGen2DbgHlcPowCtrl.up = (real32_T)FILT_IN;

  /* Product: '<S379>/Divide2' */
  r = rtb_Switch_jv * Gen2_ref_B->BusInput3.PowCtrl.rKd;

  /* DiscreteIntegrator: '<S379>/Discrete-Time Integrator1' */
  if (rtb_LogicalOperator_in || (Gen2_ref_DWork->DiscreteTimeIntegrator1_PrevR_l
       != 0)) {
    Gen2_ref_DWork->DiscreteTimeIntegrator1_DSTA_nh = 0.0;
  }

  /* Product: '<S379>/Divide3' incorporates:
   *  DiscreteIntegrator: '<S379>/Discrete-Time Integrator1'
   *  Sum: '<S379>/Sum1'
   */
  rtb_Divide3_p = (r - Gen2_ref_DWork->DiscreteTimeIntegrator1_DSTA_nh) *
    Gen2_ref_B->BusInput3.PowCtrl.rN;

  /* Delay: '<S379>/Delay2' */
  r = Gen2_ref_DWork->Delay2_DSTATE_o;

  /* MATLAB Function: '<S379>/MATLAB Function' incorporates:
   *  Constant: '<S342>/Constant'
   *  Sum: '<S379>/Sum6'
   */
  Gen2_ref_MATLABFunction_g(rtb_LogicalOperator_in, 0.0, rtb_LogicalOperator1_e,
    ((r - rtb_Switch_e3) - FILT_IN) - rtb_Divide3_p,
    &Gen2_ref_B->sf_MATLABFunction_g, &Gen2_ref_DWork->sf_MATLABFunction_g, inst);

  /* DiscreteIntegrator: '<S379>/Discrete-Time Integrator' */
  if (Gen2_ref_DWork->DiscreteTimeIntegrator_IC_LOA_g != 0) {
    Gen2_ref_DWork->DiscreteTimeIntegrator_DSTATE_f =
      Gen2_ref_B->sf_MATLABFunction_g.Y0Out;
  }

  if (Gen2_ref_B->sf_MATLABFunction_g.ireset ||
      (Gen2_ref_DWork->DiscreteTimeIntegrator_PrevR_o3 != 0)) {
    Gen2_ref_DWork->DiscreteTimeIntegrator_DSTATE_f =
      Gen2_ref_B->sf_MATLABFunction_g.Y0Out;
  }

  /* Sum: '<S379>/Sum3' incorporates:
   *  DiscreteIntegrator: '<S379>/Discrete-Time Integrator'
   *  Sum: '<S379>/Sum'
   */
  FILT_IN = ((FILT_IN + Gen2_ref_DWork->DiscreteTimeIntegrator_DSTATE_f) +
             rtb_Divide3_p) + rtb_Switch_e3;

  /* Product: '<S385>/delta rise limit' incorporates:
   *  SampleTimeMath: '<S385>/sample time'
   *
   * About '<S385>/sample time':
   *  y = K where K = ( w * Ts )
   */
  r = Gen2_ref_B->BusInput3.PowCtrl.rLam_Sr_Pos * 0.01;

  /* Delay: '<S385>/Delay' incorporates:
   *  Delay: '<S404>/Delay'
   */
  Gen2_ref_DWork->icLoad_nq = ((((Gen2_ref_PrevZCSigState->Delay_Reset_ZCE_at ==
    1) != (int32_T)rtb_LogicalOperator_in) &&
    (Gen2_ref_PrevZCSigState->Delay_Reset_ZCE_at != 3)) ||
    rtb_LogicalOperator_in || Gen2_ref_DWork->icLoad_nq);
  Gen2_ref_PrevZCSigState->Delay_Reset_ZCE_at = rtb_LogicalOperator_in;
  if (Gen2_ref_DWork->icLoad_nq) {
    Gen2_ref_DWork->Delay_DSTATE_dj = rtb_Switch_e3;
  }

  /* Switch: '<S385>/etaVolConst' */
  if (rtb_LogicalOperator_in) {
    rtb_Abs = rtb_Switch_e3;
  } else {
    rtb_Abs = FILT_IN;
  }

  /* End of Switch: '<S385>/etaVolConst' */

  /* Sum: '<S385>/Difference Inputs1' incorporates:
   *  Delay: '<S385>/Delay'
   */
  rtb_Saturation6 = rtb_Abs - Gen2_ref_DWork->Delay_DSTATE_dj;

  /* Switch: '<S386>/Switch2' incorporates:
   *  RelationalOperator: '<S386>/LowerRelop1'
   */
  if (!(rtb_Saturation6 > r)) {
    /* Product: '<S385>/delta fall limit' incorporates:
     *  SampleTimeMath: '<S385>/sample time'
     *
     * About '<S385>/sample time':
     *  y = K where K = ( w * Ts )
     */
    rtb_Abs = Gen2_ref_B->BusInput3.PowCtrl.rLam_Sr_Neg * 0.01;

    /* Switch: '<S386>/Switch' incorporates:
     *  RelationalOperator: '<S386>/UpperRelop'
     */
    if (rtb_Saturation6 < rtb_Abs) {
      r = rtb_Abs;
    } else {
      r = rtb_Saturation6;
    }

    /* End of Switch: '<S386>/Switch' */
  }

  /* End of Switch: '<S386>/Switch2' */

  /* Sum: '<S385>/Difference Inputs2' incorporates:
   *  Delay: '<S385>/Delay'
   */
  rtb_Saturation6 = r + Gen2_ref_DWork->Delay_DSTATE_dj;

  /* Switch: '<S384>/Switch2' incorporates:
   *  RelationalOperator: '<S384>/LowerRelop1'
   *  RelationalOperator: '<S384>/UpperRelop'
   *  Switch: '<S384>/Switch'
   */
  if (rtb_Saturation6 > rtb_Switch2_n5) {
    rtb_Switch2_jw = rtb_Switch2_n5;
  } else if (rtb_Saturation6 < rtb_Switch1_k) {
    /* Switch: '<S384>/Switch' */
    rtb_Switch2_jw = rtb_Switch1_k;
  } else {
    rtb_Switch2_jw = rtb_Saturation6;
  }

  /* End of Switch: '<S384>/Switch2' */

  /* Sum: '<S379>/Sum2' */
  r = rtb_Switch2_jw - FILT_IN;

  /* Product: '<S379>/Divide4' */
  r *= Gen2_ref_B->BusInput3.PowCtrl.rKaw;

  /* BusCreator: '<Root>/Bus Creator' incorporates:
   *  BusCreator: '<S379>/Bus Creator1'
   *  DataTypeConversion: '<S379>/Data Type Conversion2'
   *  DataTypeConversion: '<S379>/Data Type Conversion4'
   *  DataTypeConversion: '<S379>/Data Type Conversion7'
   *  DiscreteIntegrator: '<S379>/Discrete-Time Integrator'
   *  Outport: '<Root>/dbg'
   */
  Gen2_ref_Y->dbg.HLC.BGen2DbgHlcPowCtrl.ui = (real32_T)
    Gen2_ref_DWork->DiscreteTimeIntegrator_DSTATE_f;
  Gen2_ref_Y->dbg.HLC.BGen2DbgHlcPowCtrl.aw = (real32_T)r;
  Gen2_ref_Y->dbg.HLC.BGen2DbgHlcPowCtrl.u_unsat = (real32_T)FILT_IN;

  /* Product: '<S379>/Divide' */
  FILT_IN = rtb_Switch_jv * Gen2_ref_B->BusInput3.PowCtrl.rKi;

  /* MATLAB Function: '<S379>/MATLAB Function1' */
  Gen2_ref_MATLABFunction1(rtb_Switch2_jw, rtb_LogicalOperator1_e,
    &Gen2_ref_B->sf_MATLABFunction1_h, &Gen2_ref_DWork->sf_MATLABFunction1_h, inst);

  /* Update for DiscreteIntegrator: '<S379>/Discrete-Time Integrator1' incorporates:
   *  DiscreteIntegrator: '<S389>/Discrete-Time Integrator1'
   */
  Gen2_ref_DWork->DiscreteTimeIntegrator1_DSTA_nh += 0.01 * rtb_Divide3_p;

  /* Outputs for Atomic SubSystem: '<S343>/PID_Power' */
  Gen2_ref_DWork->DiscreteTimeIntegrator1_PrevR_l = (int8_T)
    rtb_LogicalOperator_in;

  /* End of Outputs for SubSystem: '<S343>/PID_Power' */

  /* Update for Delay: '<S379>/Delay2' */
  Gen2_ref_DWork->Delay2_DSTATE_o = Gen2_ref_B->sf_MATLABFunction1_h.LamOut;

  /* Update for DiscreteIntegrator: '<S379>/Discrete-Time Integrator' incorporates:
   *  DataTypeConversion: '<S4>/Data Type Conversion29'
   *  Sum: '<S379>/Sum4'
   *  Sum: '<S379>/Sum5'
   */
  Gen2_ref_DWork->DiscreteTimeIntegrator_IC_LOA_g = 0U;
  Gen2_ref_DWork->DiscreteTimeIntegrator_DSTATE_f +=
    (((Gen2_ref_B->BusInput.rAW_EGT_ext + rtb_Switch8) + r) + FILT_IN) * 0.01;
  Gen2_ref_DWork->DiscreteTimeIntegrator_PrevR_o3 = (int8_T)
    Gen2_ref_B->sf_MATLABFunction_g.ireset;

  /* Update for Delay: '<S385>/Delay' */
  Gen2_ref_DWork->icLoad_nq = false;
  Gen2_ref_DWork->Delay_DSTATE_dj = rtb_Saturation6;

  /* End of Outputs for SubSystem: '<S342>/PID_Power' */

  /* Gain: '<S631>/Gain2' */
  rtb_Saturation6 = 0.10471975511965977 * rtb_Switch_ks;

  /* Gain: '<S431>/Gain1' incorporates:
   *  Gain: '<S626>/Gain11'
   *  Gain: '<S631>/Gain3'
   */
  rtb_Gain1_f_tmp = 0.10471975511965977 * rtb_Switch_i5[0];

  /* Sum: '<S748>/Sum' incorporates:
   *  Gain: '<S431>/Gain1'
   *  Sum: '<S747>/Sum2'
   */
  rtb_Saturation6_tmp = rtb_Saturation6 - rtb_Gain1_f_tmp;

  /* Outputs for Atomic SubSystem: '<S747>/TON' */
  /* UnitDelay: '<S641>/Unit Delay2' */
  Gen2_ref_TON_1(Gen2_ref_DWork->UnitDelay2_DSTATE_d2,
                 Gen2_ref_B->BusInput3.SpeedCtrl.tOutOfNWindow,
                 &Gen2_ref_B->TON_d, &Gen2_ref_DWork->TON_d, inst);

  /* End of Outputs for SubSystem: '<S747>/TON' */

  /* Logic: '<S747>/Logical Operator3' incorporates:
   *  Logic: '<S747>/Logical Operator2'
   *  UnitDelay: '<S641>/Unit Delay2'
   */
  rtb_LogicalOperator3_b = (Gen2_ref_DWork->UnitDelay2_DSTATE_d2 &&
    (!Gen2_ref_B->TON_d.LogicalOperator3));

  /* Switch: '<S747>/Switch5' incorporates:
   *  Abs: '<S747>/Abs'
   *  Gain: '<S747>/Gain5'
   *  Logic: '<S747>/Logical Operator4'
   *  RelationalOperator: '<S747>/Relational Operator'
   *  Sum: '<S747>/Sum3'
   */
  if ((fabs(rtb_Saturation6_tmp * 9.5492965855137211) >
       Gen2_ref_B->BusInput3.SpeedCtrl.rOutOfNWinHys +
       Gen2_ref_B->BusInput3.SpeedCtrl.rOutOfNWindow) && rtb_LogicalOperator3_b)
  {
    rtb_bResetHlci_0 = Gen2_ref_B->BusInput3.SpeedCtrl.rOutOfNWindow;
  } else {
    rtb_bResetHlci_0 = Gen2_ref_B->BusInput3.SpeedCtrl.rThrsh_ss_int_iLQR;
  }

  /* End of Switch: '<S747>/Switch5' */

  /* RelationalOperator: '<S748>/Relational Operator' incorporates:
   *  Abs: '<S748>/Abs'
   *  Gain: '<S641>/Gain5'
   *  Sum: '<S748>/Sum'
   */
  rtb_LogicalOperator2_p1 = (fabs(rtb_Saturation6_tmp) > 0.10471975511965977 *
    rtb_bResetHlci_0);

  /* Logic: '<S748>/Logical Operator' incorporates:
   *  Logic: '<S748>/Logical Operator1'
   */
  rtb_LogicalOperator1_e = (rtb_LogicalOperator2_p1 ||
    (Gen2_ref_B->BusInput3.SpeedCtrl.bKF_act ||
     Gen2_ref_B->BusInput3.SpeedCtrl.bComModeLQR || rtb_bResetHlci));

  /* Gain: '<S641>/Gain1' */
  rtb_Switch_jv = 0.10471975511965977 *
    Gen2_ref_B->BusInput3.SpeedCtrl.rInitSpeedCtrl_iLQR;

  /* DiscreteIntegrator: '<S748>/Discrete-Time Integrator' */
  if (Gen2_ref_DWork->DiscreteTimeIntegrator_IC_LOADI != 0) {
    Gen2_ref_DWork->DiscreteTimeIntegrator_DSTATE_k = rtb_Switch_jv;
  }

  if (rtb_LogicalOperator1_e || (Gen2_ref_DWork->DiscreteTimeIntegrator_PrevRe_j
       != 0)) {
    Gen2_ref_DWork->DiscreteTimeIntegrator_DSTATE_k = rtb_Switch_jv;
  }

  /* Switch: '<S748>/Switch' incorporates:
   *  Constant: '<S748>/Constant3'
   *  DiscreteIntegrator: '<S748>/Discrete-Time Integrator'
   *  Logic: '<S748>/Logical Operator6'
   */
  if (Gen2_ref_B->BusInput3.SpeedCtrl.bTrackNbyLambda ||
      Gen2_ref_B->BusInput3.SpeedCtrl.bTrackNbyKe) {
    rtb_Switch_dhr = 0.0;
  } else {
    rtb_Switch_dhr = Gen2_ref_DWork->DiscreteTimeIntegrator_DSTATE_k;
  }

  /* End of Switch: '<S748>/Switch' */

  /* Sum: '<S641>/Sum1' */
  rtb_Sum1_l = rtb_Saturation6 + rtb_Switch_dhr;

  /* Gain: '<S431>/Gain2' */
  rtb_Gain2_cm = 1.0E-5 * rtb_Switch2_l;

  /* Switch: '<S695>/Switch2' incorporates:
   *  RelationalOperator: '<S695>/LowerRelop1'
   *  RelationalOperator: '<S695>/UpperRelop'
   *  Switch: '<S695>/Switch'
   */
  if (rtb_Gain2_cm > Gen2_ref_B->BusInput3.traj.rPr_p2s_max) {
    rtb_Abs = Gen2_ref_B->BusInput3.traj.rPr_p2s_max;
  } else if (rtb_Gain2_cm < Gen2_ref_B->BusInput3.traj.rPr_p2s_min) {
    /* Switch: '<S695>/Switch' */
    rtb_Abs = Gen2_ref_B->BusInput3.traj.rPr_p2s_min;
  } else {
    rtb_Abs = rtb_Gain2_cm;
  }

  /* End of Switch: '<S695>/Switch2' */

  /* DiscreteIntegrator: '<S748>/Discrete-Time Integrator4' */
  if (rtb_LogicalOperator1_e || (Gen2_ref_DWork->DiscreteTimeIntegrator4_PrevRes
       != 0)) {
    Gen2_ref_DWork->DiscreteTimeIntegrator4_DSTATE = 0.0;
    if (Gen2_ref_DWork->DiscreteTimeIntegrator4_DSTATE >= 0.0) {
      Gen2_ref_DWork->DiscreteTimeIntegrator4_DSTATE = 0.0;
    } else if (Gen2_ref_DWork->DiscreteTimeIntegrator4_DSTATE <= -0.3) {
      Gen2_ref_DWork->DiscreteTimeIntegrator4_DSTATE = -0.3;
    }
  }

  if (Gen2_ref_DWork->DiscreteTimeIntegrator4_DSTATE >= 0.0) {
    Gen2_ref_DWork->DiscreteTimeIntegrator4_DSTATE = 0.0;
  } else if (Gen2_ref_DWork->DiscreteTimeIntegrator4_DSTATE <= -0.3) {
    Gen2_ref_DWork->DiscreteTimeIntegrator4_DSTATE = -0.3;
  }

  /* Logic: '<S748>/Logical Operator3' incorporates:
   *  Logic: '<S748>/Logical Operator2'
   */
  rtb_LogicalOperator3_fj = (rtb_LogicalOperator2_p1 || (rtb_bResetHlci ||
    Gen2_ref_B->BusInput3.SpeedCtrl.bKF_act ||
    Gen2_ref_B->BusInput3.SpeedCtrl.bComModeLQR_boost));

  /* DiscreteIntegrator: '<S748>/Discrete-Time Integrator1' */
  if (rtb_LogicalOperator3_fj ||
      (Gen2_ref_DWork->DiscreteTimeIntegrator1_PrevRes != 0)) {
    Gen2_ref_DWork->DiscreteTimeIntegrator1_DSTATE = 0.0;
  }

  /* Sum: '<S641>/Sum2' incorporates:
   *  DiscreteIntegrator: '<S748>/Discrete-Time Integrator1'
   *  DiscreteIntegrator: '<S748>/Discrete-Time Integrator4'
   *  Sum: '<S641>/Sum4'
   *  Sum: '<S748>/Sum5'
   */
  rtb_Sum2_a_tmp = (Gen2_ref_DWork->DiscreteTimeIntegrator4_DSTATE +
                    Gen2_ref_DWork->DiscreteTimeIntegrator1_DSTATE) + rtb_Abs;

  /* Outputs for Atomic SubSystem: '<Root>/brake eff estimate' */
  /* Gain: '<S626>/Gain10' incorporates:
   *  Gain: '<S21>/Gain1'
   *  Gain: '<S631>/Gain1'
   *  Gain: '<S814>/Gain10'
   */
  rtb_Switch2_ejy_tmp = 1000.0 * Gen2_ref_B->BusInput3.leanox.rP_Eng_Frict;

  /* End of Outputs for SubSystem: '<Root>/brake eff estimate' */
  rtb_Switch2_l = rtb_Switch2_ejy_tmp;

  /* Switch: '<S626>/Switch3' */
  if (Gen2_ref_B->BusInput3.SpeedCtrl.bMeasPowKeEst) {
    rtb_bResetHlci_0 = rtb_Switch_i5[3];
  } else {
    rtb_bResetHlci_0 = rtb_Switch_bs;
  }

  /* End of Switch: '<S626>/Switch3' */

  /* Sum: '<S626>/Sum3' */
  rtb_Switch_jv = rtb_bResetHlci_0 + rtb_Switch2_l;

  /* Abs: '<S646>/Abs' incorporates:
   *  Abs: '<S694>/Abs'
   */
  r = fabs(rtb_Gain1_f_tmp);
  rtb_Switch2_l = r;

  /* Switch: '<S646>/Switch' incorporates:
   *  Constant: '<S646>/Constant2'
   *  RelationalOperator: '<S646>/Relational Operator'
   */
  if (2.2204460492503131E-16 >= rtb_Switch2_l) {
    rtb_bResetHlci_0 = 2.2204460492503131E-16;
  } else {
    rtb_bResetHlci_0 = rtb_Gain1_f_tmp;
  }

  /* End of Switch: '<S646>/Switch' */

  /* Product: '<S626>/Divide3' */
  rtb_Divide3_g = rtb_Switch_jv / rtb_bResetHlci_0;

  /* Gain: '<S431>/Gain3' incorporates:
   *  Gain: '<S628>/Gain1'
   *  Gain: '<S630>/Gain6'
   *  Gain: '<S636>/Gain1'
   *  Gain: '<S636>/Gain2'
   *  Gain: '<S636>/Gain6'
   *  Gain: '<S639>/Gain5'
   *  Switch: '<S636>/Switch6'
   */
  rtb_Gain3 = 1.0E-5 * rtb_Switch_i5[5];

  /* Saturate: '<S637>/Saturation' */
  if (Gen2_ref_B->BusInput3.PowCtrl.rLam_Start <= 1.0) {
    rtb_Saturation_o = 1.0;
  } else {
    rtb_Saturation_o = Gen2_ref_B->BusInput3.PowCtrl.rLam_Start;
  }

  /* End of Saturate: '<S637>/Saturation' */

  /* Delay: '<S637>/Resettable Delay' incorporates:
   *  Delay: '<S425>/Delay'
   */
  Gen2_ref_DWork->icLoad_ef =
    ((((Gen2_ref_PrevZCSigState->ResettableDelay_Reset_ZCE_m == 1) != (int32_T)
       rtb_bResetHlci) && (Gen2_ref_PrevZCSigState->ResettableDelay_Reset_ZCE_m
       != 3)) || rtb_bResetHlci || Gen2_ref_DWork->icLoad_ef);
  Gen2_ref_PrevZCSigState->ResettableDelay_Reset_ZCE_m = rtb_bResetHlci;
  if (Gen2_ref_DWork->icLoad_ef) {
    Gen2_ref_DWork->ResettableDelay_DSTATE_i = rtb_Saturation_o;
  }

  rtb_Switch_jv = Gen2_ref_DWork->ResettableDelay_DSTATE_i;

  /* Abs: '<S736>/Abs' */
  rtb_Switch2_l = fabs(rtb_Product1_aq);

  /* Switch: '<S736>/Switch' incorporates:
   *  Constant: '<S736>/Constant2'
   *  RelationalOperator: '<S736>/Relational Operator'
   */
  if (2.2204460492503131E-16 >= rtb_Switch2_l) {
    rtb_Product1_aq = 2.2204460492503131E-16;
  }

  /* End of Switch: '<S736>/Switch' */

  /* Product: '<S639>/Product1' */
  rtb_Product1_aq = rtb_Switch_i5[3] / rtb_Product1_aq;

  /* Outputs for Atomic SubSystem: '<S737>/Filter' */
  /* DiscreteIntegrator: '<S743>/Discrete-Time Integrator' incorporates:
   *  Logic: '<S743>/Logical Operator'
   */
  if (Gen2_ref_DWork->DiscreteTimeIntegrator_IC_LOA_m != 0) {
    Gen2_ref_DWork->DiscreteTimeIntegrator_DSTATE_n = rtb_Product1_aq;
  }

  if (rtb_bResetHlci || (Gen2_ref_DWork->DiscreteTimeIntegrator_PrevR_kx != 0))
  {
    Gen2_ref_DWork->DiscreteTimeIntegrator_DSTATE_n = rtb_Product1_aq;
  }

  /* Switch: '<S743>/Switch' incorporates:
   *  DiscreteIntegrator: '<S743>/Discrete-Time Integrator'
   */
  rtb_Switch_nb = Gen2_ref_DWork->DiscreteTimeIntegrator_DSTATE_n;

  /* Update for DiscreteIntegrator: '<S743>/Discrete-Time Integrator' incorporates:
   *  Logic: '<S743>/Logical Operator'
   *  Product: '<S743>/Divide4'
   *  Sum: '<S743>/Sum4'
   */
  Gen2_ref_DWork->DiscreteTimeIntegrator_IC_LOA_m = 0U;
  Gen2_ref_DWork->DiscreteTimeIntegrator_DSTATE_n += (rtb_Product1_aq -
    Gen2_ref_DWork->DiscreteTimeIntegrator_DSTATE_n) / 0.1 * 0.01;
  Gen2_ref_DWork->DiscreteTimeIntegrator_PrevR_kx = (int8_T)rtb_bResetHlci;

  /* End of Outputs for SubSystem: '<S737>/Filter' */

  /* Switch: '<S737>/Switch3' */
  if (Gen2_ref_B->BusInput3.SpeedCtrl.bGS_D_iLQR) {
    /* Saturate: '<S737>/Saturation' */
    if (rtb_Switch_nb > 1.0) {
      rtb_Product1_aq = 1.0;
    } else if (rtb_Switch_nb < 0.0) {
      rtb_Product1_aq = 0.0;
    } else {
      rtb_Product1_aq = rtb_Switch_nb;
    }

    /* End of Saturate: '<S737>/Saturation' */

    /* S-Function (sfix_look1_dyn): '<S737>/gain scheduling D' */
    /* Dynamic Look-Up Table Block: '<S737>/gain scheduling D'
     * Input0  Data Type:  Floating Point real_T
     * Input1  Data Type:  Floating Point real_T
     * Input2  Data Type:  Floating Point real_T
     * Output0 Data Type:  Floating Point real_T
     * Lookup Method: Linear_Endpoint
     *
     */
    LookUp_real_T_real_T( &(rtb_gainschedulingD),
                         &Gen2_ref_B->BusInput3.SpeedCtrl.refPoint_iLQR_D_y[0],
                         rtb_Product1_aq,
                         &Gen2_ref_B->BusInput3.SpeedCtrl.refPoint_iLQR_D_x[0],
                         5U, inst);
    rtb_Switch_nb = rtb_gainschedulingD;
  } else {
    rtb_Switch_nb = Gen2_ref_B->BusInput3.SpeedCtrl.rD_iLQR;
  }

  /* End of Switch: '<S737>/Switch3' */

  /* Abs: '<S742>/Abs' incorporates:
   *  Abs: '<S731>/Abs'
   */
  rtb_Switch_dz_tmp = fabs(Gen2_ref_B->BusInput3.eng.Ts);
  rtb_Switch2_l = rtb_Switch_dz_tmp;

  /* Switch: '<S742>/Switch' incorporates:
   *  Constant: '<S742>/Constant2'
   *  RelationalOperator: '<S742>/Relational Operator'
   */
  if (2.2204460492503131E-16 >= rtb_Switch2_l) {
    rtb_bResetHlci_0 = 2.2204460492503131E-16;
  } else {
    rtb_bResetHlci_0 = Gen2_ref_B->BusInput3.eng.Ts;
  }

  /* End of Switch: '<S742>/Switch' */

  /* Product: '<S737>/Product1' incorporates:
   *  Product: '<S737>/Product'
   *  Rounding: '<S737>/Rounding Function'
   */
  rtb_Product1_b4 = floor(rtb_Switch_nb / rtb_bResetHlci_0) *
    Gen2_ref_B->BusInput3.eng.Ts;

  /* Switch: '<S731>/Switch' incorporates:
   *  Constant: '<S731>/Constant2'
   *  RelationalOperator: '<S731>/Relational Operator'
   */
  if (0.001 >= rtb_Switch_dz_tmp) {
    rtb_bResetHlci_0 = 0.001;
  } else {
    rtb_bResetHlci_0 = Gen2_ref_B->BusInput3.eng.Ts;
  }

  /* End of Switch: '<S731>/Switch' */

  /* DataTypeConversion: '<S637>/Data Type Conversion' incorporates:
   *  Product: '<S637>/Divide'
   */
  rtb_bResetHlci_0 = floor(rtb_Product1_b4 / rtb_bResetHlci_0);
  if (rtIsNaN(rtb_bResetHlci_0) || rtIsInf(rtb_bResetHlci_0)) {
    rtb_bResetHlci_0 = 0.0;
  } else {
    rtb_bResetHlci_0 = fmod(rtb_bResetHlci_0, 65536.0);
  }

  rtb_DataTypeConversion_l = (uint16_T)(rtb_bResetHlci_0 < 0.0 ? (int32_T)
    (uint16_T)-(int16_T)(uint16_T)-rtb_bResetHlci_0 : (int32_T)(uint16_T)
    rtb_bResetHlci_0);

  /* End of DataTypeConversion: '<S637>/Data Type Conversion' */

  /* Delay: '<S637>/Variable Integer Delay' incorporates:
   *  Delay: '<S425>/Delay'
   *  Delay: '<S637>/Resettable Delay'
   */
  if ((((Gen2_ref_PrevZCSigState->VariableIntegerDelay_Reset_ZCE == 1) !=
        (int32_T)rtb_bResetHlci) &&
       (Gen2_ref_PrevZCSigState->VariableIntegerDelay_Reset_ZCE != 3)) ||
      rtb_bResetHlci) {
    Gen2_ref_DWork->icLoad_b = true;
    Gen2_ref_DWork->CircBufIdx = 0U;
  }

  Gen2_ref_PrevZCSigState->VariableIntegerDelay_Reset_ZCE = rtb_bResetHlci;
  if (Gen2_ref_DWork->icLoad_b) {
    for (i = 0; i < 200; i++) {
      Gen2_ref_DWork->VariableIntegerDelay_DSTATE[i] = rtb_Saturation_o;
    }
  }

  if (rtb_DataTypeConversion_l <= 0) {
    rtb_VariableIntegerDelay = Gen2_ref_DWork->ResettableDelay_DSTATE_i;
  } else {
    if (rtb_DataTypeConversion_l > 200) {
      rtb_DataTypeConversion_l = 200U;
    }

    if (rtb_DataTypeConversion_l <= Gen2_ref_DWork->CircBufIdx) {
      rtb_DataTypeConversion_l = (uint16_T)((uint32_T)Gen2_ref_DWork->CircBufIdx
        - rtb_DataTypeConversion_l);
    } else {
      rtb_DataTypeConversion_l = (uint16_T)((uint16_T)((uint32_T)
        Gen2_ref_DWork->CircBufIdx - rtb_DataTypeConversion_l) + 200U);
    }

    rtb_VariableIntegerDelay = Gen2_ref_DWork->
      VariableIntegerDelay_DSTATE[rtb_DataTypeConversion_l];
  }

  /* End of Delay: '<S637>/Variable Integer Delay' */

  /* Gain: '<S639>/Gain5' */
  rtb_Product1_aq = rtb_Gain3;

  /* Switch: '<S740>/Switch3' */
  if (Gen2_ref_B->BusInput3.SpeedCtrl.bGS_T_Lam_iLQR) {
    /* S-Function (sfix_look1_dyn): '<S740>/gain scheduling Tlam' */
    /* Dynamic Look-Up Table Block: '<S740>/gain scheduling Tlam'
     * Input0  Data Type:  Floating Point real_T
     * Input1  Data Type:  Floating Point real_T
     * Input2  Data Type:  Floating Point real_T
     * Output0 Data Type:  Floating Point real_T
     * Lookup Method: Linear_Endpoint
     *
     */
    LookUp_real_T_real_T( &(rtb_gainschedulingTlam),
                         &Gen2_ref_B->BusInput3.SpeedCtrl.refPoint_iLQR_Tlam_y[0],
                         rtb_Product1_aq,
                         &Gen2_ref_B->BusInput3.SpeedCtrl.refPoint_iLQR_Tlam_x[0],
                         6U, inst);
    rtb_Switch_nb = rtb_gainschedulingTlam;
  } else {
    rtb_Switch_nb = Gen2_ref_B->BusInput3.SpeedCtrl.rTi_Lam_iLQR;
  }

  /* End of Switch: '<S740>/Switch3' */

  /* UnitDelay: '<S628>/Unit Delay1' */
  rtb_Switch2_l = Gen2_ref_DWork->UnitDelay1_DSTATE_a;

  /* Switch: '<S740>/Switch4' incorporates:
   *  Constant: '<S740>/Constant5'
   */
  if (!Gen2_ref_B->BusInput3.SpeedCtrl.bAddTi_Tlam) {
    rtb_Switch2_l = 0.0;
  }

  /* End of Switch: '<S740>/Switch4' */

  /* Sum: '<S740>/Sum2' */
  rtb_Sum2_kg = rtb_Switch_nb + rtb_Switch2_l;

  /* Outputs for Atomic SubSystem: '<S637>/Filter' */
  Gen2_ref_Pd_filt(rtb_VariableIntegerDelay, rtb_Sum2_kg, rtb_Saturation_o,
                   rtb_bResetHlci, &Gen2_ref_B->Filter_bd,
                   &Gen2_ref_DWork->Filter_bd, inst);

  /* End of Outputs for SubSystem: '<S637>/Filter' */

  /* Sum: '<S626>/Sum4' incorporates:
   *  Constant: '<S626>/it_offset_ref2'
   *  Product: '<S626>/Divide5'
   */
  rtb_Switch_nb = Gen2_ref_B->Filter_bd.Switch * rtb_Sum1_idx_2 + 1.0;

  /* Abs: '<S647>/Abs' */
  rtb_Switch2_l = fabs(rtb_Switch_nb);

  /* Switch: '<S647>/Switch' incorporates:
   *  Constant: '<S647>/Constant2'
   *  RelationalOperator: '<S647>/Relational Operator'
   */
  if (2.2204460492503131E-16 >= rtb_Switch2_l) {
    rtb_Switch_nb = 2.2204460492503131E-16;
  }

  /* End of Switch: '<S647>/Switch' */

  /* Product: '<S626>/Divide4' */
  rtb_Switch_nb = rtb_Gain3 / rtb_Switch_nb;

  /* Abs: '<S648>/Abs' */
  rtb_Switch2_l = fabs(rtb_Switch_nb);

  /* Switch: '<S648>/Switch' incorporates:
   *  Constant: '<S648>/Constant2'
   *  RelationalOperator: '<S648>/Relational Operator'
   */
  if (2.2204460492503131E-16 >= rtb_Switch2_l) {
    rtb_Switch_nb = 2.2204460492503131E-16;
  }

  /* End of Switch: '<S648>/Switch' */

  /* Outputs for Atomic SubSystem: '<S626>/Filter1' */
  /* Product: '<S626>/Divide11' */
  Gen2_ref_N_TC_HP_filt(rtb_Divide3_g / rtb_Switch_nb,
                        Gen2_ref_B->BusInput3.SpeedCtrl.rTiFKeEst,
                        rtb_bResetHlci, &Gen2_ref_B->Filter1_o,
                        &Gen2_ref_DWork->Filter1_o, inst);

  /* End of Outputs for SubSystem: '<S626>/Filter1' */

  /* Delay: '<S625>/Delay' */
  rtb_Switch2_l = Gen2_ref_DWork->Delay_DSTATE_k;

  /* Switch: '<S625>/Switch' incorporates:
   *  Constant: '<S625>/R_air'
   */
  if (!Gen2_ref_B->BusInput3.SpeedCtrl.bUseRgasEst) {
    rtb_Switch2_l = 287.15;
  }

  /* End of Switch: '<S625>/Switch' */

  /* Abs: '<S643>/Abs' incorporates:
   *  Abs: '<S149>/Abs'
   *  Abs: '<S273>/Abs'
   *  Abs: '<S289>/Abs'
   */
  rtb_bResetHlci_0 = fabs(Gen2_ref_B->T2s_filt.Switch);

  /* Switch: '<S643>/Switch' incorporates:
   *  Abs: '<S643>/Abs'
   *  Constant: '<S643>/Constant2'
   *  RelationalOperator: '<S643>/Relational Operator'
   */
  if (2.2204460492503131E-16 >= rtb_bResetHlci_0) {
    delta_y = 2.2204460492503131E-16;
  } else {
    delta_y = Gen2_ref_B->T2s_filt.Switch;
  }

  /* End of Switch: '<S643>/Switch' */

  /* Switch: '<S642>/Switch' incorporates:
   *  Abs: '<S642>/Abs'
   *  Constant: '<S642>/Constant2'
   *  RelationalOperator: '<S642>/Relational Operator'
   */
  if (2.2204460492503131E-16 >= fabs(rtb_Switch2_l)) {
    rtb_Switch2_l = 2.2204460492503131E-16;
  }

  /* End of Switch: '<S642>/Switch' */

  /* Gain: '<S625>/Gain1' incorporates:
   *  Gain: '<S625>/Gain2'
   *  Product: '<S625>/Divide3'
   */
  rtb_VariableIntegerDelay = Gen2_ref_B->BusInput3.eng.rVol_Hub_Eng / delta_y *
    rtb_etaVolConst_lt * rtb_etaBreakConst * rtb_Sum1_idx_3 / rtb_Switch2_l *
    0.079577471545947673 * 100000.0;

  /* Product: '<S8>/Product1' incorporates:
   *  DataTypeConversion: '<S8>/Data Type Conversion2'
   */
  rtb_Product1_fu = (real_T)Gen2_ref_B->BusInput3.SkipF.bSF_ON * rtb_Switch2_ba;

  /* Saturate: '<S625>/Saturation' */
  if (Gen2_ref_B->BusInput3.eng.rNum_Cyl_Eng <= 1.0) {
    delta_y = 1.0;
  } else {
    delta_y = Gen2_ref_B->BusInput3.eng.rNum_Cyl_Eng;
  }

  /* End of Saturate: '<S625>/Saturation' */

  /* Product: '<S625>/Divide1' */
  u0 = Gen2_ref_B->BusInput3.SpeedCtrl.rK_skip_iLQR / delta_y * rtb_Product1_fu;

  /* Saturate: '<S625>/Saturation1' */
  if (u0 > 1.0) {
    u0 = 1.0;
  } else if (u0 < 0.0) {
    u0 = 0.0;
  }

  /* End of Saturate: '<S625>/Saturation1' */

  /* Product: '<S625>/Product' incorporates:
   *  Constant: '<S625>/it_offset_ref2'
   *  Sum: '<S625>/Sum3'
   */
  rtb_Switch_nb = (1.0 - u0) * rtb_VariableIntegerDelay;

  /* Abs: '<S670>/Abs' */
  rtb_Switch2_l = fabs(rtb_Switch_nb);

  /* Switch: '<S670>/Switch' incorporates:
   *  Constant: '<S670>/Constant2'
   *  RelationalOperator: '<S670>/Relational Operator'
   */
  if (2.2204460492503131E-16 >= rtb_Switch2_l) {
    delta_y = 2.2204460492503131E-16;
  } else {
    delta_y = rtb_Switch_nb;
  }

  /* End of Switch: '<S670>/Switch' */

  /* Product: '<S666>/Product1' */
  rtb_Divide3_g = Gen2_ref_B->Filter1_o.Switch / delta_y;

  /* Gain: '<S630>/Gain6' */
  rtb_Gain6_b = rtb_Gain3;

  /* Logic: '<S666>/Logical Operator3' incorporates:
   *  Logic: '<S714>/Logical Operator3'
   *  Logic: '<S830>/Logical Operator3'
   */
  rtb_LogicalOperator2_l = !Gen2_ref_B->BusInput3.SpeedCtrl.bKeAdaptON;

  /* Logic: '<S666>/Logical Operator2' incorporates:
   *  Logic: '<S666>/Logical Operator3'
   */
  rtb_LogicalOperator_f = (rtb_bResetHlci || rtb_LogicalOperator2_l);

  /* Delay: '<S666>/Resettable Delay' */
  Gen2_ref_DWork->icLoad_i0 = ((rtb_LogicalOperator_f &&
    (Gen2_ref_PrevZCSigState->ResettableDelay_Reset_ZCE_a != 1)) ||
    Gen2_ref_DWork->icLoad_i0);
  Gen2_ref_PrevZCSigState->ResettableDelay_Reset_ZCE_a = rtb_LogicalOperator_f;
  for (i = 0; i < 13; i++) {
    if (Gen2_ref_DWork->icLoad_i0) {
      Gen2_ref_DWork->ResettableDelay_DSTATE_a[i] =
        Gen2_ref_B->BusInput3.SpeedCtrl.refPoint_iLQR_Keng_y[i];
    }

    rtb_ResettableDelay_br[i] = Gen2_ref_DWork->ResettableDelay_DSTATE_a[i];
  }

  /* End of Delay: '<S666>/Resettable Delay' */

  /* S-Function (sfix_look1_dyn): '<S666>/gain scheduling Keng1' */
  /* Dynamic Look-Up Table Block: '<S666>/gain scheduling Keng1'
   * Input0  Data Type:  Floating Point real_T
   * Input1  Data Type:  Floating Point real_T
   * Input2  Data Type:  Floating Point real_T
   * Output0 Data Type:  Floating Point real_T
   * Lookup Method: Linear_Endpoint
   *
   */
  LookUp_real_T_real_T( &(rtb_gainschedulingKeng1), &rtb_ResettableDelay_br[0],
                       rtb_Gain6_b,
                       &Gen2_ref_B->BusInput3.SpeedCtrl.refPoint_iLQR_Keng_x[0],
                       12U, inst);

  /* Outputs for Atomic SubSystem: '<S667>/TP' */
  /* UnitDelay: '<S667>/Unit Delay2' incorporates:
   *  SignalConversion generated from: '<S667>/Bus Selector1'
   */
  Gen2_ref_TP(Gen2_ref_DWork->UnitDelay2_DSTATE_n,
              Gen2_ref_B->BusInput3.SpeedCtrl.rTp_KeEst_reset,
              &Gen2_ref_B->TP_p2, &Gen2_ref_DWork->TP_p2, inst);

  /* End of Outputs for SubSystem: '<S667>/TP' */

  /* Outputs for Atomic SubSystem: '<S667>/TON1' */
  Gen2_ref_TON_1(Gen2_ref_DWork->UnitDelay2_DSTATE_n,
                 Gen2_ref_B->BusInput3.SpeedCtrl.tOutOfNWindow,
                 &Gen2_ref_B->TON1, &Gen2_ref_DWork->TON1, inst);

  /* End of Outputs for SubSystem: '<S667>/TON1' */

  /* Switch: '<S667>/Switch2' incorporates:
   *  Constant: '<S667>/Constant1'
   *  Switch: '<S667>/Switch'
   */
  if (Gen2_ref_B->BusInput3.SpeedCtrl.bKeEstResetOFF) {
    rtb_Switch2_ij = false;
  } else if (Gen2_ref_B->BusInput3.SpeedCtrl.bKeEstreset_TP) {
    /* Switch: '<S667>/Switch' */
    rtb_Switch2_ij = Gen2_ref_B->TP_p2.LogicalOperator1;
  } else {
    /* Switch: '<S667>/Switch' incorporates:
     *  Logic: '<S667>/Logical Operator4'
     *  Logic: '<S667>/Logical Operator5'
     *  UnitDelay: '<S667>/Unit Delay2'
     */
    rtb_Switch2_ij = (Gen2_ref_DWork->UnitDelay2_DSTATE_n &&
                      (!Gen2_ref_B->TON1.LogicalOperator3));
  }

  /* End of Switch: '<S667>/Switch2' */

  /* Outputs for Atomic SubSystem: '<S667>/TP1' */
  /* UnitDelay: '<S667>/Unit Delay2' incorporates:
   *  SignalConversion generated from: '<S667>/Bus Selector9'
   */
  Gen2_ref_TP(Gen2_ref_DWork->UnitDelay2_DSTATE_n,
              Gen2_ref_B->BusInput3.SpeedCtrl.rT_KeEstIncreaseTiF,
              &Gen2_ref_B->TP1_c, &Gen2_ref_DWork->TP1_c, inst);

  /* End of Outputs for SubSystem: '<S667>/TP1' */

  /* UnitDelay: '<S667>/Unit Delay1' */
  rtb_Switch2_l = Gen2_ref_DWork->UnitDelay1_DSTATE_e;

  /* DataTypeConversion: '<S667>/Data Type Conversion' */
  delta_y = floor(rtb_Switch2_l);
  if (rtIsNaN(delta_y) || rtIsInf(delta_y)) {
    delta_y = 0.0;
  } else {
    delta_y = fmod(delta_y, 65536.0);
  }

  /* Outputs for Atomic SubSystem: '<S667>/TOF' */
  /* RelationalOperator: '<S667>/Relational Operator' incorporates:
   *  DataTypeConversion: '<S667>/Data Type Conversion'
   */
  Gen2_ref_TOF(((delta_y < 0.0 ? (int32_T)(int16_T)-(int16_T)(uint16_T)-delta_y :
                 (int32_T)(int16_T)(uint16_T)delta_y) > 0),
               Gen2_ref_B->BusInput3.SpeedCtrl.rTof_KeEstPause_SkipF,
               &Gen2_ref_B->TOF_g, &Gen2_ref_DWork->TOF_g, inst);

  /* End of Outputs for SubSystem: '<S667>/TOF' */

  /* Switch: '<S667>/Switch3' incorporates:
   *  Constant: '<S667>/Constant2'
   *  Switch: '<S667>/Switch1'
   */
  if (Gen2_ref_B->BusInput3.SpeedCtrl.bKeEstIncreaseTiFOFF) {
    rtb_Switch3_of = false;
  } else if (Gen2_ref_B->BusInput3.SpeedCtrl.bKeEstPause_SkipF) {
    /* Switch: '<S667>/Switch1' incorporates:
     *  Logic: '<S667>/Logical Operator3'
     */
    rtb_Switch3_of = (Gen2_ref_B->TP1_c.LogicalOperator1 ||
                      Gen2_ref_B->TOF_g.LogicalOperator1);
  } else {
    /* Switch: '<S667>/Switch1' */
    rtb_Switch3_of = Gen2_ref_B->TP1_c.LogicalOperator1;
  }

  /* End of Switch: '<S667>/Switch3' */

  /* Outputs for Atomic SubSystem: '<S666>/Ke Map Update' */
  Gen2_ref_KeMapUpdate(rtb_Divide3_g, rtb_bResetHlci, rtb_gainschedulingKeng1,
                       rtb_Switch3_of, rtb_Switch2_ij, &Gen2_ref_B->BusInput3,
                       &Gen2_ref_B->KeMapUpdate, &Gen2_ref_DWork->KeMapUpdate, inst);

  /* End of Outputs for SubSystem: '<S666>/Ke Map Update' */

  /* Switch: '<S666>/Switch1' incorporates:
   *  Logic: '<S666>/Logical Operator4'
   */
  if (!Gen2_ref_B->BusInput3.SpeedCtrl.bActKeEst2Dof) {
    rtb_Switch1_ep = rtb_Divide3_g;
  } else {
    rtb_Switch1_ep = Gen2_ref_B->KeMapUpdate.Sum1;
  }

  /* End of Switch: '<S666>/Switch1' */

  /* Logic: '<S630>/Logical Operator1' incorporates:
   *  Logic: '<S630>/Logical Operator2'
   *  Logic: '<S636>/Logical Operator5'
   */
  rtb_LogicalOperator5_g_tmp = (Gen2_ref_B->BusInput3.SpeedCtrl.bKF_act &&
    (!Gen2_ref_B->BusInput3.SpeedCtrl.bKeMap4KF));

  /* Outputs for Atomic SubSystem: '<S630>/Filter' */
  /* Constant: '<S630>/Constant3' incorporates:
   *  Logic: '<S630>/Logical Operator1'
   *  Logic: '<S630>/Logical Operator3'
   *  Logic: '<S630>/Logical Operator4'
   */
  Gen2_ref_Filter(1.0, rtb_Switch1_ep, ((!rtb_LogicalOperator5_g_tmp) ||
    rtb_bResetHlci), &Gen2_ref_B->Filter_nk, &Gen2_ref_ConstB.Filter_nk,
                  &Gen2_ref_DWork->Filter_nk, inst);

  /* End of Outputs for SubSystem: '<S630>/Filter' */

  /* Gain: '<S636>/Gain6' */
  rtb_Gain6_jx = rtb_Gain3;

  /* Logic: '<S431>/Logical Operator' */
  rtb_LogicalOperator_hi = (rtb_bResetHlci ||
    Gen2_ref_B->BusInput3.SpeedCtrl.bActKeEstMapUpdate);

  /* Logic: '<S714>/Logical Operator2' incorporates:
   *  Logic: '<S715>/Logical Operator2'
   */
  rtb_LogicalOperator2_k_tmp = (rtb_LogicalOperator_hi || rtb_LogicalOperator2_l);

  /* Delay: '<S714>/Resettable Delay1' incorporates:
   *  Logic: '<S714>/Logical Operator2'
   */
  Gen2_ref_DWork->icLoad_np = ((rtb_LogicalOperator2_k_tmp &&
    (Gen2_ref_PrevZCSigState->ResettableDelay1_Reset_ZCE != 1)) ||
    Gen2_ref_DWork->icLoad_np);
  Gen2_ref_PrevZCSigState->ResettableDelay1_Reset_ZCE =
    rtb_LogicalOperator2_k_tmp;

  /* Delay: '<S714>/Resettable Delay' incorporates:
   *  Logic: '<S714>/Logical Operator2'
   */
  Gen2_ref_DWork->icLoad_j = ((rtb_LogicalOperator2_k_tmp &&
    (Gen2_ref_PrevZCSigState->ResettableDelay_Reset_ZCE_e != 1)) ||
    Gen2_ref_DWork->icLoad_j);
  Gen2_ref_PrevZCSigState->ResettableDelay_Reset_ZCE_e =
    rtb_LogicalOperator2_k_tmp;
  for (i = 0; i < 13; i++) {
    /* Delay: '<S714>/Resettable Delay1' */
    if (Gen2_ref_DWork->icLoad_np) {
      Gen2_ref_DWork->ResettableDelay1_DSTATE[i] =
        Gen2_ref_B->BusInput3.SpeedCtrl.refPoint_iLQR_Keng_y[i];
    }

    /* Delay: '<S714>/Resettable Delay' */
    if (Gen2_ref_DWork->icLoad_j) {
      Gen2_ref_DWork->ResettableDelay_DSTATE_m[i] =
        Gen2_ref_B->BusInput3.SpeedCtrl.refPoint_iLQR_Keng_y[i];
    }

    /* Switch: '<S714>/Switch' incorporates:
     *  Delay: '<S714>/Resettable Delay'
     *  Delay: '<S714>/Resettable Delay1'
     *  UnitDelay: '<S714>/Unit Delay1'
     */
    if (Gen2_ref_DWork->UnitDelay1_DSTATE_o) {
      rtb_ResettableDelay_br[i] = Gen2_ref_DWork->ResettableDelay1_DSTATE[i];
    } else {
      rtb_ResettableDelay_br[i] = Gen2_ref_DWork->ResettableDelay_DSTATE_m[i];
    }

    /* End of Switch: '<S714>/Switch' */
  }

  /* S-Function (sfix_look1_dyn): '<S714>/gain scheduling Keng1' */
  /* Dynamic Look-Up Table Block: '<S714>/gain scheduling Keng1'
   * Input0  Data Type:  Floating Point real_T
   * Input1  Data Type:  Floating Point real_T
   * Input2  Data Type:  Floating Point real_T
   * Output0 Data Type:  Floating Point real_T
   * Lookup Method: Linear_Endpoint
   *
   */
  LookUp_real_T_real_T( &(rtb_Switch2_l), &rtb_ResettableDelay_br[0],
                       rtb_Gain6_jx,
                       &Gen2_ref_B->BusInput3.SpeedCtrl.refPoint_iLQR_Keng_x[0],
                       12U, inst);

  /* DiscreteIntegrator: '<S714>/Discrete-Time Integrator' incorporates:
   *  Logic: '<S714>/Logical Operator2'
   */
  if (rtb_LogicalOperator2_k_tmp ||
      (Gen2_ref_DWork->DiscreteTimeIntegrator_PrevRe_o != 0)) {
    Gen2_ref_DWork->DiscreteTimeIntegrator_DSTATE_l = 0.0;
  }

  /* Sum: '<S714>/Sum' incorporates:
   *  DiscreteIntegrator: '<S714>/Discrete-Time Integrator'
   */
  rtb_Sum_ig = rtb_Switch2_l + Gen2_ref_DWork->DiscreteTimeIntegrator_DSTATE_l;

  /* Abs: '<S712>/Abs' */
  rtb_Switch2_l = rtb_Product1_e_tmp;

  /* Switch: '<S712>/Switch' incorporates:
   *  Constant: '<S712>/Constant2'
   *  RelationalOperator: '<S712>/Relational Operator'
   */
  if (2.2204460492503131E-16 >= rtb_Switch2_l) {
    delta_y = 2.2204460492503131E-16;
  } else {
    delta_y = Gen2_ref_B->BusInput3.eng.rP_Nom;
  }

  /* End of Switch: '<S712>/Switch' */

  /* Product: '<S636>/Divide' */
  rtb_Switch2_l = rtb_Switch_i5[3] / delta_y;

  /* Gain: '<S636>/Gain7' */
  rtb_Gain7 = 0.001 * rtb_Switch2_l;

  /* RelationalOperator: '<S636>/Relational Operator' */
  rtb_RelationalOperator_ok = (rtb_Gain7 >
    Gen2_ref_B->BusInput3.SpeedCtrl.rMinPow_p2sGSC);

  /* Delay: '<S715>/Resettable Delay1' incorporates:
   *  Logic: '<S714>/Logical Operator2'
   */
  Gen2_ref_DWork->icLoad_a = ((rtb_LogicalOperator2_k_tmp &&
    (Gen2_ref_PrevZCSigState->ResettableDelay1_Reset_ZCE_g != 1)) ||
    Gen2_ref_DWork->icLoad_a);
  Gen2_ref_PrevZCSigState->ResettableDelay1_Reset_ZCE_g =
    rtb_LogicalOperator2_k_tmp;

  /* Delay: '<S715>/Resettable Delay' incorporates:
   *  Logic: '<S714>/Logical Operator2'
   */
  Gen2_ref_DWork->icLoad_m3 = ((rtb_LogicalOperator2_k_tmp &&
    (Gen2_ref_PrevZCSigState->ResettableDelay_Reset_ZCE_b != 1)) ||
    Gen2_ref_DWork->icLoad_m3);
  Gen2_ref_PrevZCSigState->ResettableDelay_Reset_ZCE_b =
    rtb_LogicalOperator2_k_tmp;
  for (i = 0; i < 7; i++) {
    /* Delay: '<S715>/Resettable Delay1' */
    if (Gen2_ref_DWork->icLoad_a) {
      Gen2_ref_DWork->ResettableDelay1_DSTATE_e[i] =
        Gen2_ref_B->BusInput3.SpeedCtrl.refPoint_iLQR_KengPOW_y[i];
    }

    /* Delay: '<S715>/Resettable Delay' */
    if (Gen2_ref_DWork->icLoad_m3) {
      Gen2_ref_DWork->ResettableDelay_DSTATE_e[i] =
        Gen2_ref_B->BusInput3.SpeedCtrl.refPoint_iLQR_KengPOW_y[i];
    }

    /* Switch: '<S715>/Switch' incorporates:
     *  Delay: '<S715>/Resettable Delay'
     *  Delay: '<S715>/Resettable Delay1'
     *  UnitDelay: '<S715>/Unit Delay1'
     */
    if (Gen2_ref_DWork->UnitDelay1_DSTATE_j) {
      rtb_Switch_dau[i] = Gen2_ref_DWork->ResettableDelay1_DSTATE_e[i];
    } else {
      rtb_Switch_dau[i] = Gen2_ref_DWork->ResettableDelay_DSTATE_e[i];
    }

    /* End of Switch: '<S715>/Switch' */
  }

  /* S-Function (sfix_look1_dyn): '<S715>/gain scheduling Keng1' */
  /* Dynamic Look-Up Table Block: '<S715>/gain scheduling Keng1'
   * Input0  Data Type:  Floating Point real_T
   * Input1  Data Type:  Floating Point real_T
   * Input2  Data Type:  Floating Point real_T
   * Output0 Data Type:  Floating Point real_T
   * Lookup Method: Linear_Endpoint
   *
   */
  LookUp_real_T_real_T( &(rtb_Switch2_l), &rtb_Switch_dau[0], rtb_Gain7,
                       &Gen2_ref_B->BusInput3.SpeedCtrl.refPoint_iLQR_KengPOW_x
                       [0], 6U, inst);

  /* DiscreteIntegrator: '<S715>/Discrete-Time Integrator' */
  if (rtb_LogicalOperator2_k_tmp ||
      (Gen2_ref_DWork->DiscreteTimeIntegrator_PrevRe_n != 0)) {
    Gen2_ref_DWork->DiscreteTimeIntegrator_DSTATE_e = 0.0;
  }

  /* Sum: '<S715>/Sum' incorporates:
   *  DiscreteIntegrator: '<S715>/Discrete-Time Integrator'
   */
  rtb_Sum_gb = rtb_Switch2_l + Gen2_ref_DWork->DiscreteTimeIntegrator_DSTATE_e;

  /* Switch: '<S636>/Switch2' */
  if (Gen2_ref_B->BusInput3.SpeedCtrl.bGS_Ke_iLQR) {
    /* Switch: '<S636>/Switch1' incorporates:
     *  Switch: '<S636>/Switch4'
     */
    if (rtb_RelationalOperator_ok) {
      /* Switch: '<S636>/Switch5' */
      if (Gen2_ref_B->BusInput3.SpeedCtrl.bKeAdaptON) {
        rtb_Divide3_g = rtb_Sum_ig;
      } else {
        /* S-Function (sfix_look1_dyn): '<S636>/gain scheduling Keng' */
        /* Dynamic Look-Up Table Block: '<S636>/gain scheduling Keng'
         * Input0  Data Type:  Floating Point real_T
         * Input1  Data Type:  Floating Point real_T
         * Input2  Data Type:  Floating Point real_T
         * Output0 Data Type:  Floating Point real_T
         * Lookup Method: Linear_Endpoint
         *
         */
        LookUp_real_T_real_T( &(rtb_gainschedulingKeng),
                             &Gen2_ref_B->BusInput3.SpeedCtrl.refPoint_iLQR_Keng_y
                             [0], rtb_Gain6_jx,
                             &Gen2_ref_B->BusInput3.SpeedCtrl.refPoint_iLQR_Keng_x
                             [0], 12U, inst);
        rtb_Divide3_g = rtb_gainschedulingKeng;
      }

      /* End of Switch: '<S636>/Switch5' */
    } else if (Gen2_ref_B->BusInput3.SpeedCtrl.bKeAdaptON) {
      /* Switch: '<S636>/Switch4' */
      rtb_Divide3_g = rtb_Sum_gb;
    } else {
      /* S-Function (sfix_look1_dyn): '<S636>/gain scheduling KengPOW' incorporates:
       *  Switch: '<S636>/Switch4'
       */
      /* Dynamic Look-Up Table Block: '<S636>/gain scheduling KengPOW'
       * Input0  Data Type:  Floating Point real_T
       * Input1  Data Type:  Floating Point real_T
       * Input2  Data Type:  Floating Point real_T
       * Output0 Data Type:  Floating Point real_T
       * Lookup Method: Linear_Endpoint
       *
       */
      LookUp_real_T_real_T( &(rtb_gainschedulingKengPOW),
                           &Gen2_ref_B->BusInput3.SpeedCtrl.refPoint_iLQR_KengPOW_y
                           [0], rtb_Gain7,
                           &Gen2_ref_B->BusInput3.SpeedCtrl.refPoint_iLQR_KengPOW_x
                           [0], 6U, inst);

      /* Switch: '<S636>/Switch4' */
      rtb_Divide3_g = rtb_gainschedulingKengPOW;
    }

    /* End of Switch: '<S636>/Switch1' */
  } else {
    rtb_Divide3_g = Gen2_ref_B->BusInput3.SpeedCtrl.rFactKe_iLQR;
  }

  /* End of Switch: '<S636>/Switch2' */

  /* Outputs for Atomic SubSystem: '<S636>/Filter' */
  /* Constant: '<S636>/Constant3' incorporates:
   *  Logic: '<S636>/Logical Operator3'
   *  Logic: '<S636>/Logical Operator4'
   */
  Gen2_ref_Filter(1.0, rtb_Divide3_g, ((!rtb_LogicalOperator5_g_tmp) ||
    rtb_LogicalOperator_hi), &Gen2_ref_B->Filter_m, &Gen2_ref_ConstB.Filter_m,
                  &Gen2_ref_DWork->Filter_m, inst);

  /* End of Outputs for SubSystem: '<S636>/Filter' */

  /* Switch: '<S431>/Switch2' incorporates:
   *  Switch: '<S636>/Switch3'
   */
  if (Gen2_ref_B->BusInput3.SpeedCtrl.bActKeEstMapUpdate) {
    /* Switch: '<S630>/Switch3' incorporates:
     *  Logic: '<S630>/Logical Operator1'
     */
    if (rtb_LogicalOperator5_g_tmp) {
      rtb_Switch2_l = Gen2_ref_B->Filter_nk.Switch;
    } else {
      rtb_Switch2_l = rtb_Switch1_ep;
    }

    /* End of Switch: '<S630>/Switch3' */
  } else if (rtb_LogicalOperator5_g_tmp) {
    /* Switch: '<S636>/Switch3' */
    rtb_Switch2_l = Gen2_ref_B->Filter_m.Switch;
  } else {
    rtb_Switch2_l = rtb_Divide3_g;
  }

  /* End of Switch: '<S431>/Switch2' */

  /* Product: '<S431>/Product' */
  rtb_Product_o = rtb_Switch2_l * rtb_Switch_nb;

  /* Gain: '<S631>/Gain1' */
  rtb_Switch2_l = rtb_Switch2_ejy_tmp;

  /* Switch: '<S692>/Switch' incorporates:
   *  Abs: '<S692>/Abs'
   *  Constant: '<S692>/Constant2'
   *  RelationalOperator: '<S692>/Relational Operator'
   */
  if (2.2204460492503131E-16 >= fabs(rtb_Saturation6)) {
    delta_y = 2.2204460492503131E-16;
  } else {
    delta_y = rtb_Saturation6;
  }

  /* End of Switch: '<S692>/Switch' */

  /* Product: '<S631>/Divide' incorporates:
   *  Sum: '<S631>/Sum'
   */
  rtb_Divide_i1 = (rtb_Switch_bs + rtb_Switch2_l) / delta_y;

  /* Switch: '<S693>/Switch' incorporates:
   *  Abs: '<S693>/Abs'
   *  Constant: '<S693>/Constant2'
   *  RelationalOperator: '<S693>/Relational Operator'
   */
  if (2.2204460492503131E-16 >= fabs(rtb_Divide_i1)) {
    delta_y = 2.2204460492503131E-16;
  } else {
    delta_y = rtb_Divide_i1;
  }

  /* End of Switch: '<S693>/Switch' */

  /* Switch: '<S631>/Switch1' incorporates:
   *  Constant: '<S631>/Constant3'
   */
  if (Gen2_ref_B->BusInput3.SpeedCtrl.bExternalOffsetON) {
    FILT_IN = rtb_Sum4_ny;
  } else {
    FILT_IN = 0.0;
  }

  /* End of Switch: '<S631>/Switch1' */

  /* Sum: '<S631>/Sum2' incorporates:
   *  Constant: '<S631>/it_offset_ref1'
   *  Product: '<S631>/Divide1'
   *  Product: '<S631>/Divide2'
   *  Sum: '<S631>/Sum1'
   */
  rtb_Gain2_cm = (rtb_Gain2_cm * rtb_Product_o / delta_y - 1.0) / rtb_Sum1_idx_2
    + FILT_IN;

  /* Switch: '<S696>/Switch2' incorporates:
   *  RelationalOperator: '<S696>/LowerRelop1'
   *  RelationalOperator: '<S696>/UpperRelop'
   *  Switch: '<S696>/Switch'
   */
  if (rtb_Gain2_cm > rtb_Switch2_n5) {
    rtb_Switch2_c4 = rtb_Switch2_n5;
  } else if (rtb_Gain2_cm < rtb_Switch1_k) {
    /* Switch: '<S696>/Switch' */
    rtb_Switch2_c4 = rtb_Switch1_k;
  } else {
    rtb_Switch2_c4 = rtb_Gain2_cm;
  }

  /* End of Switch: '<S696>/Switch2' */

  /* DiscreteIntegrator: '<S748>/Discrete-Time Integrator3' */
  if (rtb_LogicalOperator1_e || (Gen2_ref_DWork->DiscreteTimeIntegrator3_PrevRes
       != 0)) {
    Gen2_ref_DWork->DiscreteTimeIntegrator3_DSTATE = 0.0;
  }

  /* Switch: '<S748>/Switch1' incorporates:
   *  DiscreteIntegrator: '<S748>/Discrete-Time Integrator'
   *  DiscreteIntegrator: '<S748>/Discrete-Time Integrator3'
   *  Gain: '<S748>/Gain'
   *  Logic: '<S748>/Logical Operator4'
   *  Logic: '<S748>/Logical Operator5'
   */
  if (Gen2_ref_B->BusInput3.SpeedCtrl.bTrackNbyLambda &&
      (!Gen2_ref_B->BusInput3.SpeedCtrl.bTrackNbyKe)) {
    rtb_Gain2_cm = -0.01 * Gen2_ref_DWork->DiscreteTimeIntegrator_DSTATE_k;
  } else {
    rtb_Gain2_cm = Gen2_ref_DWork->DiscreteTimeIntegrator3_DSTATE;
  }

  /* End of Switch: '<S748>/Switch1' */

  /* Sum: '<S641>/Sum6' incorporates:
   *  Sum: '<S641>/Sum5'
   */
  rtb_Sum6_o_tmp = rtb_Switch2_c4 + rtb_Gain2_cm;

  /* Switch: '<S697>/Switch2' incorporates:
   *  Constant: '<S631>/it_offset_ref'
   *  RelationalOperator: '<S697>/LowerRelop1'
   *  RelationalOperator: '<S697>/UpperRelop'
   *  Switch: '<S697>/Switch'
   */
  if (0.0 > Gen2_ref_B->BusInput3.SpeedCtrl.rDeltaZZP_max_iLQR) {
    rtb_Switch2_oou = Gen2_ref_B->BusInput3.SpeedCtrl.rDeltaZZP_max_iLQR;
  } else if (0.0 < Gen2_ref_B->BusInput3.SpeedCtrl.rDeltaZZP_min_iLQR) {
    /* Switch: '<S697>/Switch' */
    rtb_Switch2_oou = Gen2_ref_B->BusInput3.SpeedCtrl.rDeltaZZP_min_iLQR;
  } else {
    rtb_Switch2_oou = 0.0;
  }

  /* End of Switch: '<S697>/Switch2' */

  /* Switch: '<S431>/Switch9' incorporates:
   *  Constant: '<S431>/Constant6'
   *  Rounding: '<S629>/Rounding Function'
   */
  if (Gen2_ref_B->BusInput3.SpeedCtrl.bSF_OFF_iLQR) {
    rtb_Switch9_k = 0.0;
  } else {
    /* Sum: '<S629>/Sum1' */
    rtb_Gain2_cm = Gen2_ref_B->BusInput3.SkipF.rP_max_1 -
      Gen2_ref_B->BusInput3.SkipF.rP_max_0;

    /* Switch: '<S662>/Switch' incorporates:
     *  Abs: '<S662>/Abs'
     *  Constant: '<S662>/Constant2'
     *  RelationalOperator: '<S662>/Relational Operator'
     */
    if (2.2204460492503131E-16 >= fabs(rtb_Gain2_cm)) {
      rtb_Gain2_cm = 2.2204460492503131E-16;
    }

    /* End of Switch: '<S662>/Switch' */

    /* Sum: '<S629>/Sum3' incorporates:
     *  Gain: '<S629>/Gain'
     *  Product: '<S629>/Divide'
     *  Sum: '<S629>/Sum'
     *  Sum: '<S629>/Sum2'
     */
    rtb_Gain2_cm = (0.001 * rtb_Switch_bs - Gen2_ref_B->BusInput3.SkipF.rP_max_0)
      * (Gen2_ref_B->BusInput3.SkipF.rNum_max_P1 -
         Gen2_ref_B->BusInput3.SkipF.rNum_max_P0) / rtb_Gain2_cm +
      Gen2_ref_B->BusInput3.SkipF.rNum_max_P0;

    /* Switch: '<S663>/Switch2' incorporates:
     *  Constant: '<S629>/Constant5'
     *  RelationalOperator: '<S663>/LowerRelop1'
     *  RelationalOperator: '<S663>/UpperRelop'
     *  Switch: '<S663>/Switch'
     */
    if (rtb_Gain2_cm > Gen2_ref_B->BusInput3.SkipF.rNum_max) {
      rtb_Gain2_cm = Gen2_ref_B->BusInput3.SkipF.rNum_max;
    } else if (rtb_Gain2_cm < 0.0) {
      /* Switch: '<S663>/Switch' incorporates:
       *  Constant: '<S629>/Constant5'
       */
      rtb_Gain2_cm = 0.0;
    }

    /* End of Switch: '<S663>/Switch2' */
    rtb_Switch9_k = rt_roundd_snf(rtb_Gain2_cm, inst);
  }

  /* End of Switch: '<S431>/Switch9' */

  /* Switch: '<S698>/Switch2' incorporates:
   *  Constant: '<S431>/Nskip_min'
   *  RelationalOperator: '<S698>/LowerRelop1'
   *  RelationalOperator: '<S698>/UpperRelop'
   *  Switch: '<S698>/Switch'
   */
  if (rtb_Product1_fu > rtb_Switch9_k) {
    rtb_Gain2_cm = rtb_Switch9_k;
  } else if (rtb_Product1_fu < 0.0) {
    /* Switch: '<S698>/Switch' incorporates:
     *  Constant: '<S431>/Nskip_min'
     */
    rtb_Gain2_cm = 0.0;
  } else {
    rtb_Gain2_cm = rtb_Product1_fu;
  }

  /* End of Switch: '<S698>/Switch2' */

  /* DiscreteIntegrator: '<S748>/Discrete-Time Integrator2' */
  if (rtb_LogicalOperator1_e || (Gen2_ref_DWork->DiscreteTimeIntegrator2_PrevRes
       != 0)) {
    Gen2_ref_DWork->DiscreteTimeIntegrator2_DSTATE = 0.0;
  }

  /* Sum: '<S641>/Sum3' incorporates:
   *  DiscreteIntegrator: '<S748>/Discrete-Time Integrator2'
   */
  rtb_Sum3_o = rtb_Gain2_cm + Gen2_ref_DWork->DiscreteTimeIntegrator2_DSTATE;

  /* Delay: '<S431>/Delay' incorporates:
   *  SignalConversion generated from: '<S431>/Delay'
   */
  if (Gen2_ref_DWork->icLoad_b3) {
    Gen2_ref_DWork->Delay_DSTATE_ba[0] = rtb_Sum2_a_tmp;
    Gen2_ref_DWork->Delay_DSTATE_ba[1] = rtb_Sum6_o_tmp;
    Gen2_ref_DWork->Delay_DSTATE_ba[2] = rtb_Switch2_oou;
    Gen2_ref_DWork->Delay_DSTATE_ba[3] = rtb_Sum3_o;
  }

  /* Switch: '<S694>/Switch' incorporates:
   *  Constant: '<S694>/Constant2'
   *  RelationalOperator: '<S694>/Relational Operator'
   */
  if (2.2204460492503131E-16 >= r) {
    delta_y = 2.2204460492503131E-16;
  } else {
    delta_y = rtb_Gain1_f_tmp;
  }

  /* End of Switch: '<S694>/Switch' */

  /* Product: '<S631>/Divide3' incorporates:
   *  Sum: '<S631>/Sum3'
   */
  rtb_Divide3_ep = (rtb_Switch_i5[3] + rtb_Switch2_l) / delta_y;

  /* Switch: '<S738>/Switch' */
  if (Gen2_ref_B->BusInput3.SpeedCtrl.bGS_iLQR_R1) {
    /* S-Function (sfix_look1_dyn): '<S738>/Lookup Table Dynamic' */
    /* Dynamic Look-Up Table Block: '<S738>/Lookup Table Dynamic'
     * Input0  Data Type:  Floating Point real_T
     * Input1  Data Type:  Floating Point real_T
     * Input2  Data Type:  Floating Point real_T
     * Output0 Data Type:  Floating Point real_T
     * Saturation Mode: Saturate
     * Lookup Method: Linear_Endpoint
     *
     */
    LookUp_real_T_real_T_SAT( &(rtb_LookupTableDynamic_l),
      &Gen2_ref_B->BusInput3.SpeedCtrl.refPoint_iLQR_R1_y[0], rtb_Product1_aq,
      &Gen2_ref_B->BusInput3.SpeedCtrl.refPoint_iLQR_RQT_x[0], 5U, inst);
    rtb_Divide3_i0[0] = Gen2_ref_B->BusInput3.SpeedCtrl.rR_iLQR[0];
    rtb_Divide3_i0[1] = rtb_LookupTableDynamic_l;
    rtb_Divide3_i0[2] = Gen2_ref_B->BusInput3.SpeedCtrl.rR_iLQR[2];
    rtb_Divide3_i0[3] = Gen2_ref_B->BusInput3.SpeedCtrl.rR_iLQR[3];
  } else {
    rtb_Divide3_i0[0] = Gen2_ref_B->BusInput3.SpeedCtrl.rR_iLQR[0];
    rtb_Divide3_i0[1] = Gen2_ref_B->BusInput3.SpeedCtrl.rR_iLQR[1];
    rtb_Divide3_i0[2] = Gen2_ref_B->BusInput3.SpeedCtrl.rR_iLQR[2];
    rtb_Divide3_i0[3] = Gen2_ref_B->BusInput3.SpeedCtrl.rR_iLQR[3];
  }

  /* End of Switch: '<S738>/Switch' */

  /* Product: '<S738>/Product' */
  rtb_Product_m[0] = Gen2_ref_B->BusInput3.SpeedCtrl.rFactorRilqr *
    rtb_Divide3_i0[0];
  rtb_Product_m[1] = Gen2_ref_B->BusInput3.SpeedCtrl.rFactorRilqr *
    rtb_Divide3_i0[1];
  rtb_Product_m[2] = Gen2_ref_B->BusInput3.SpeedCtrl.rFactorRilqr *
    rtb_Divide3_i0[2];
  rtb_Product_m[3] = Gen2_ref_B->BusInput3.SpeedCtrl.rFactorRilqr *
    rtb_Divide3_i0[3];

  /* Switch: '<S738>/Switch1' */
  if (Gen2_ref_B->BusInput3.SpeedCtrl.bGS_iLQR_Q0) {
    /* S-Function (sfix_look1_dyn): '<S738>/Lookup Table Dynamic1' */
    /* Dynamic Look-Up Table Block: '<S738>/Lookup Table Dynamic1'
     * Input0  Data Type:  Floating Point real_T
     * Input1  Data Type:  Floating Point real_T
     * Input2  Data Type:  Floating Point real_T
     * Output0 Data Type:  Floating Point real_T
     * Saturation Mode: Saturate
     * Lookup Method: Linear_Endpoint
     *
     */
    LookUp_real_T_real_T_SAT( &(rtb_LookupTableDynamic1_g),
      &Gen2_ref_B->BusInput3.SpeedCtrl.refPoint_iLQR_Q0_y[0], rtb_Product1_aq,
      &Gen2_ref_B->BusInput3.SpeedCtrl.refPoint_iLQR_RQT_x[0], 5U, inst);
    rtb_Switch1_cl[0] = rtb_LookupTableDynamic1_g;
    rtb_Switch1_cl[1] = Gen2_ref_B->BusInput3.SpeedCtrl.rQ_iLQR[1];
    rtb_Switch1_cl[2] = Gen2_ref_B->BusInput3.SpeedCtrl.rQ_iLQR[2];
  } else {
    rtb_Switch1_cl[0] = Gen2_ref_B->BusInput3.SpeedCtrl.rQ_iLQR[0];
    rtb_Switch1_cl[1] = Gen2_ref_B->BusInput3.SpeedCtrl.rQ_iLQR[1];
    rtb_Switch1_cl[2] = Gen2_ref_B->BusInput3.SpeedCtrl.rQ_iLQR[2];
  }

  /* End of Switch: '<S738>/Switch1' */

  /* Switch: '<S739>/Switch' */
  if (Gen2_ref_B->BusInput3.SpeedCtrl.bGS_iLQR_TBDC) {
    /* S-Function (sfix_look1_dyn): '<S739>/Lookup Table Dynamic2' */
    /* Dynamic Look-Up Table Block: '<S739>/Lookup Table Dynamic2'
     * Input0  Data Type:  Floating Point real_T
     * Input1  Data Type:  Floating Point real_T
     * Input2  Data Type:  Floating Point real_T
     * Output0 Data Type:  Floating Point real_T
     * Saturation Mode: Saturate
     * Lookup Method: Linear_Endpoint
     *
     */
    LookUp_real_T_real_T_SAT( &(rtb_LookupTableDynamic2_h),
      &Gen2_ref_B->BusInput3.SpeedCtrl.refPoint_TBDC_y[0], rtb_Product1_aq,
      &Gen2_ref_B->BusInput3.SpeedCtrl.refPoint_iLQR_RQT_x[0], 5U, inst);
    rtb_Switch_czo = rtb_LookupTableDynamic2_h;
  } else {
    rtb_Switch_czo = Gen2_ref_B->BusInput3.SpeedCtrl.rTi_BDC_iLQR;
  }

  /* End of Switch: '<S739>/Switch' */

  /* S-Function (sfix_look1_dyn): '<S639>/Lookup Table Dynamic1' */
  /* Dynamic Look-Up Table Block: '<S639>/Lookup Table Dynamic1'
   * Input0  Data Type:  Floating Point real_T
   * Input1  Data Type:  Floating Point real_T
   * Input2  Data Type:  Floating Point real_T
   * Output0 Data Type:  Floating Point real_T
   * Lookup Method: Linear_Endpoint
   *
   */
  LookUp_real_T_real_T( &(rtb_kappa0),
                       &Gen2_ref_B->BusInput3.SpeedCtrl.rKappa0_iLQR_y[0],
                       rtb_Product1_aq,
                       &Gen2_ref_B->BusInput3.SpeedCtrl.rKappa0_iLQR_x[0], 4U, inst);

  /* Switch: '<S605>/Switch' incorporates:
   *  Constant: '<S605>/Constant2'
   *  RelationalOperator: '<S605>/Relational Operator'
   */
  if (2.2204460492503131E-16 >= rtb_Product1_e_tmp) {
    delta_y = 2.2204460492503131E-16;
  } else {
    delta_y = Gen2_ref_B->BusInput3.eng.rP_Nom;
  }

  /* End of Switch: '<S605>/Switch' */

  /* Gain: '<S581>/Gain6' incorporates:
   *  Gain: '<S581>/Gain3'
   *  Product: '<S581>/Divide3'
   */
  rtb_Product1_aq = -(0.001 * rtb_Gain1_fr / delta_y);

  /* Saturate: '<S581>/Saturation' */
  if (rtb_Product1_aq > 1000.0) {
    rtb_Product1_aq = 1000.0;
  } else if (rtb_Product1_aq < 0.0) {
    rtb_Product1_aq = 0.0;
  }

  /* End of Saturate: '<S581>/Saturation' */

  /* Gain: '<S581>/Gain1' */
  rtb_Switch2_l = -rtb_Divide_mr_tmp;

  /* Saturate: '<S581>/Saturation1' */
  if (rtb_Switch2_l > 1000.0) {
    rtb_Divide3_g = 1000.0;
  } else if (rtb_Switch2_l < 0.0) {
    rtb_Divide3_g = 0.0;
  } else {
    rtb_Divide3_g = rtb_Switch2_l;
  }

  /* End of Saturate: '<S581>/Saturation1' */

  /* Product: '<S581>/Divide2' */
  rtb_Switch2_l = rtb_Divide3_g * Gen2_ref_B->BusInput3.SkipF.rKp_skiplevel;

  /* Sum: '<S581>/Sum1' incorporates:
   *  Product: '<S581>/Divide1'
   */
  rtb_rSkip_level = rtb_Product1_aq * Gen2_ref_B->BusInput3.SkipF.rKd_skiplevel
    + rtb_Switch2_l;

  /* Switch: '<S606>/Switch1' incorporates:
   *  Constant: '<S606>/Constant3'
   *  Logic: '<S581>/Logical Operator1'
   *  RelationalOperator: '<S581>/Relational Operator'
   *  RelationalOperator: '<S581>/Relational Operator1'
   *  RelationalOperator: '<S581>/Relational Operator2'
   *  UnitDelay: '<S606>/Unit Delay'
   */
  if (rtb_Divide3_g >= Gen2_ref_B->BusInput3.SkipF.rN_limit_skip_off) {
    rtb_LogicalOperator1_ja = ((rtb_Divide3_g >=
      Gen2_ref_B->BusInput3.SkipF.rN_limit_skip_on) || (rtb_Product1_aq >=
      Gen2_ref_B->BusInput3.SkipF.rProt_limit_skip_on) ||
      Gen2_ref_DWork->UnitDelay_DSTATE_ma);
  } else {
    rtb_LogicalOperator1_ja = false;
  }

  /* End of Switch: '<S606>/Switch1' */

  /* Switch: '<S581>/Switch1' incorporates:
   *  Constant: '<S581>/  2'
   */
  if (rtb_LogicalOperator1_ja) {
    rtb_Switch2_l = rtb_rSkip_level;
  } else {
    rtb_Switch2_l = 0.0;
  }

  /* End of Switch: '<S581>/Switch1' */

  /* UnitDelay: '<S608>/Unit Delay' */
  rtb_LogicalOperator5 = Gen2_ref_DWork->TP_state;

  /* Switch: '<S604>/Switch' incorporates:
   *  Abs: '<S604>/Abs'
   *  Constant: '<S604>/Constant2'
   *  RelationalOperator: '<S604>/Relational Operator'
   */
  if (2.2204460492503131E-16 >= fabs(Gen2_ref_B->BusInput3.eng.rN_Nom)) {
    rtb_Saturation_o = 2.2204460492503131E-16;
  } else {
    rtb_Saturation_o = Gen2_ref_B->BusInput3.eng.rN_Nom;
  }

  /* End of Switch: '<S604>/Switch' */

  /* Outputs for Atomic SubSystem: '<S608>/SkipPulseWaitTP' */
  /* RelationalOperator: '<S611>/FixPt Relational Operator' incorporates:
   *  Constant: '<S608>/Constant'
   *  DataTypeConversion: '<S581>/Data Type Conversion8'
   *  Gain: '<S581>/ to Hz1'
   *  Gain: '<S581>/Hz to cycle period3'
   *  Product: '<S581>/Divide5'
   *  Sum: '<S608>/Sum'
   *  UnitDelay: '<S608>/Unit Delay'
   *  UnitDelay: '<S611>/Delay Input1'
   */
  Gen2_ref_TP(((int32_T)Gen2_ref_DWork->TP_state < (int32_T)
               Gen2_ref_DWork->DelayInput1_DSTATE), 2.0 * (60.0 * ((real_T)
    Gen2_ref_B->BusInput3.SkipF.iNr_cycles_ignON / rtb_Saturation_o)) - 0.01,
              &Gen2_ref_B->SkipPulseWaitTP, &Gen2_ref_DWork->SkipPulseWaitTP, inst);

  /* End of Outputs for SubSystem: '<S608>/SkipPulseWaitTP' */

  /* Logic: '<S581>/Logical Operator2' */
  rtb_LogicalOperator2_ov = !rtb_LogicalOperator1_ja;

  /* Logic: '<S608>/Logical Operator4' incorporates:
   *  Delay: '<S608>/Delay to avoid alg.loop'
   */
  rtb_LogicalOperator4_m5 = (Gen2_ref_DWork->Delaytoavoidalgloop_DSTATE ||
    Gen2_ref_B->SkipPulseWaitTP.LogicalOperator1 || rtb_LogicalOperator2_ov);

  /* DiscreteIntegrator: '<S608>/Discrete-Time Integrator' */
  if (rtb_LogicalOperator4_m5 ||
      (Gen2_ref_DWork->DiscreteTimeIntegrator_PrevRe_m != 0)) {
    Gen2_ref_DWork->DiscreteTimeIntegrator_DSTAT_h5 = 0.0;
  }

  /* Logic: '<S608>/Logical Operator1' incorporates:
   *  DiscreteIntegrator: '<S608>/Discrete-Time Integrator'
   *  Logic: '<S608>/Logical Operator2'
   *  Logic: '<S608>/Logical Operator3'
   *  RelationalOperator: '<S608>/Relational Operator'
   */
  rtb_LogicalOperator1_pa = ((Gen2_ref_DWork->DiscreteTimeIntegrator_DSTAT_h5 >=
    Gen2_ref_B->BusInput3.SkipF.rThrsh_PulseGenerator_trigger) &&
    (!Gen2_ref_B->SkipPulseWaitTP.LogicalOperator1) && (!rtb_LogicalOperator2_ov));

  /* Switch: '<S581>/Switch' incorporates:
   *  RelationalOperator: '<S603>/FixPt Relational Operator'
   *  UnitDelay: '<S581>/Unit Delay'
   *  UnitDelay: '<S603>/Delay Input1'
   */
  if ((int32_T)rtb_LogicalOperator1_pa > (int32_T)
      Gen2_ref_DWork->DelayInput1_DSTATE_n) {
    rtb_Product1_aq = rtb_Switch2_l;
  } else {
    rtb_Product1_aq = Gen2_ref_DWork->UnitDelay_DSTATE_f;
  }

  /* End of Switch: '<S581>/Switch' */

  /* MinMax: '<S581>/MinMax' */
  if ((rtb_Switch2_l >= rtb_Product1_aq) || rtIsNaN(rtb_Product1_aq)) {
    rtb_Product1_aq = rtb_Switch2_l;
  }

  /* End of MinMax: '<S581>/MinMax' */

  /* Product: '<S581>/Product' */
  rtb_Divide3_g = rtb_Product1_aq * (real_T)rtb_LogicalOperator1_pa;

  /* Switch: '<S607>/Switch2' incorporates:
   *  Constant: '<S581>/  10'
   *  RelationalOperator: '<S607>/LowerRelop1'
   *  RelationalOperator: '<S607>/UpperRelop'
   *  Switch: '<S607>/Switch'
   */
  if (rtb_Divide3_g > Gen2_ref_B->BusInput3.eng.rNum_Cyl_Eng) {
    rtb_Divide1_h4 = Gen2_ref_B->BusInput3.eng.rNum_Cyl_Eng;
  } else if (rtb_Divide3_g < 0.0) {
    /* Switch: '<S607>/Switch' incorporates:
     *  Constant: '<S581>/  10'
     */
    rtb_Divide1_h4 = 0.0;
  } else {
    rtb_Divide1_h4 = rtb_Divide3_g;
  }

  /* End of Switch: '<S607>/Switch2' */

  /* Quantizer: '<S581>/Quantizer1' */
  rtb_Divide1_f1_tmp = rt_roundd_snf(rtb_Divide1_h4, inst);

  /* Gain: '<S582>/Gain1' incorporates:
   *  Gain: '<S581>/Gain1'
   */
  rtb_Gain1_o = -rtb_Divide_mr_tmp;

  /* Switch: '<S622>/Switch2' incorporates:
   *  Constant: '<S582>/  1'
   *  RelationalOperator: '<S622>/LowerRelop1'
   *  RelationalOperator: '<S622>/UpperRelop'
   *  Switch: '<S622>/Switch'
   */
  if (rtb_Gain1_o > 500.0) {
    rtb_Divide1_h4 = 500.0;
  } else if (rtb_Gain1_o < Gen2_ref_B->BusInput3.SkipF.rN_LevelNskip) {
    /* Switch: '<S622>/Switch' */
    rtb_Divide1_h4 = Gen2_ref_B->BusInput3.SkipF.rN_LevelNskip;
  } else {
    rtb_Divide1_h4 = rtb_Gain1_o;
  }

  /* End of Switch: '<S622>/Switch2' */

  /* Product: '<S582>/Product1' incorporates:
   *  Sum: '<S582>/Sum3'
   */
  rtb_Divide3_g = (rtb_Divide1_h4 - Gen2_ref_B->BusInput3.SkipF.rN_LevelNskip) *
    Gen2_ref_B->BusInput3.SkipF.rKp;

  /* MATLAB Function: '<S582>/MATLAB Function1' */
  Gen2_ref_MATLABFunction_n(rtb_Divide3_g, Gen2_ref_B->BusInput3.SkipF.rHy_eps,
    &Gen2_ref_B->sf_MATLABFunction1_e, &Gen2_ref_DWork->sf_MATLABFunction1_e, inst);

  /* Gain: '<S582>/Gain3' */
  rtb_Divide1_h4 = -Gen2_ref_B->BusInput3.SkipF.rN_LevelNskip_lowN;

  /* Switch: '<S623>/Switch2' incorporates:
   *  RelationalOperator: '<S623>/LowerRelop1'
   */
  if (!(rtb_Gain1_o > rtb_Divide1_h4)) {
    /* Switch: '<S623>/Switch' incorporates:
     *  Constant: '<S582>/  2'
     *  RelationalOperator: '<S623>/UpperRelop'
     */
    if (rtb_Gain1_o < -500.0) {
      rtb_Divide1_h4 = -500.0;
    } else {
      rtb_Divide1_h4 = rtb_Gain1_o;
    }

    /* End of Switch: '<S623>/Switch' */
  }

  /* End of Switch: '<S623>/Switch2' */

  /* Product: '<S582>/Product2' incorporates:
   *  Sum: '<S582>/Sum8'
   */
  rtb_Gain1_o = (Gen2_ref_B->BusInput3.SkipF.rN_LevelNskip_lowN + rtb_Divide1_h4)
    * Gen2_ref_B->BusInput3.SkipF.rKp_lowN;

  /* MATLAB Function: '<S582>/MATLAB Function' */
  Gen2_ref_MATLABFunction_n(rtb_Gain1_o, Gen2_ref_B->BusInput3.SkipF.rHy_eps,
    &Gen2_ref_B->sf_MATLABFunction_k, &Gen2_ref_DWork->sf_MATLABFunction_k, inst);

  /* Switch: '<S429>/Switch5' incorporates:
   *  Sum: '<S582>/Sum1'
   *  Switch: '<S582>/Switch1'
   */
  if (Gen2_ref_B->BusInput3.SkipF.bSkipfire_pulse_active) {
    /* Switch: '<S581>/Switch4' incorporates:
     *  Constant: '<S581>/  16'
     *  DataTypeConversion: '<S581>/Data Type Conversion6'
     */
    if (Gen2_ref_B->BusInput3.SkipF.bSkipfire_pulse_active) {
      rtb_Switch5_iq = (real32_T)rtb_Divide1_f1_tmp;
    } else {
      rtb_Switch5_iq = 0.0;
    }

    /* End of Switch: '<S581>/Switch4' */
  } else {
    if (Gen2_ref_B->BusInput3.SkipF.bSFroundFB_ON) {
      /* Switch: '<S582>/Switch1' */
      rtb_Divide3_g = Gen2_ref_B->sf_MATLABFunction1_e.y;
    }

    /* Switch: '<S582>/Switch' */
    if (Gen2_ref_B->BusInput3.SkipF.bSFroundFB_ON_lowN) {
      rtb_Gain1_o = Gen2_ref_B->sf_MATLABFunction_k.y;
    }

    /* End of Switch: '<S582>/Switch' */
    rtb_Switch5_iq = rtb_Divide3_g + rtb_Gain1_o;
  }

  /* End of Switch: '<S429>/Switch5' */

  /* Switch: '<S632>/Switch2' incorporates:
   *  Constant: '<S431>/Constant'
   *  RelationalOperator: '<S632>/LowerRelop1'
   *  RelationalOperator: '<S632>/UpperRelop'
   *  Switch: '<S632>/Switch'
   */
  if (rtb_Switch5_iq > Gen2_ref_B->BusInput3.eng.rNum_Cyl_Eng) {
    rtb_Divide3_g = Gen2_ref_B->BusInput3.eng.rNum_Cyl_Eng;
  } else if (rtb_Switch5_iq < 0.0) {
    /* Switch: '<S632>/Switch' incorporates:
     *  Constant: '<S431>/Constant'
     */
    rtb_Divide3_g = 0.0;
  } else {
    rtb_Divide3_g = rtb_Switch5_iq;
  }

  /* End of Switch: '<S632>/Switch2' */

  /* Outputs for Atomic SubSystem: '<S716>/TON' */
  /* Logic: '<S716>/Logical Operator1' incorporates:
   *  Logic: '<S716>/Logical Operator2'
   *  UnitDelay: '<S716>/Unit Delay3'
   */
  Gen2_ref_TON_1(((!Gen2_ref_DWork->UnitDelay3_DSTATE_go) &&
                  Gen2_ref_B->TON2.LogicalOperator3),
                 Gen2_ref_B->BusInput3.SpeedCtrl.rT_x_dist1_map_update,
                 &Gen2_ref_B->TON_j, &Gen2_ref_DWork->TON_j, inst);

  /* End of Outputs for SubSystem: '<S716>/TON' */

  /* Gain: '<S636>/Gain1' */
  rtb_Divide1_h4 = rtb_Gain3;

  /* UnitDelay: '<S716>/Unit Delay1' */
  for (i = 0; i < 13; i++) {
    rtb_Switch3_je[i] = Gen2_ref_DWork->UnitDelay1_DSTATE_f[i];
  }

  /* End of UnitDelay: '<S716>/Unit Delay1' */

  /* S-Function (sfix_look1_dyn): '<S716>/gain scheduling x_dist1' */
  /* Dynamic Look-Up Table Block: '<S716>/gain scheduling x_dist1'
   * Input0  Data Type:  Floating Point real_T
   * Input1  Data Type:  Floating Point real_T
   * Input2  Data Type:  Floating Point real_T
   * Output0 Data Type:  Floating Point real_T
   * Lookup Method: Linear_Endpoint
   *
   */
  LookUp_real_T_real_T( &(rtb_Switch2_l), &rtb_Switch3_je[0], rtb_Divide1_h4,
                       &Gen2_ref_B->BusInput3.SpeedCtrl.refPoint_KF_x_dist1_x[0],
                       12U, inst);

  /* Switch: '<S716>/Switch1' incorporates:
   *  Constant: '<S716>/Constant2'
   *  UnitDelay: '<S716>/Unit Delay2'
   */
  if (Gen2_ref_B->BusInput3.SpeedCtrl.bKF_GS_xdist1) {
    delta_y = Gen2_ref_DWork->UnitDelay2_DSTATE_m;
  } else {
    delta_y = 0.0;
  }

  /* End of Switch: '<S716>/Switch1' */

  /* Sum: '<S716>/Sum' */
  rtb_Gain1_o = delta_y + rtb_Switch2_l;

  /* MATLAB Function: '<S716>/MATLAB Function' incorporates:
   *  DataTypeConversion: '<S716>/Data Type Conversion6'
   */
  if ((!Gen2_ref_DWork->y_map_not_empty) || rtb_LogicalOperator_hi) {
    Gen2_ref_DWork->y_map_not_empty = true;
    for (i = 0; i < 13; i++) {
      Gen2_ref_DWork->y_map[i] =
        Gen2_ref_B->BusInput3.SpeedCtrl.refPoint_KF_x_dist1_y[i];
      Gen2_ref_DWork->x_map[i] =
        Gen2_ref_B->BusInput3.SpeedCtrl.refPoint_KF_x_dist1_x[i];
    }
  }

  u0 = Gen2_ref_minimum(Gen2_ref_DWork->x_map, inst);
  if ((u0 >= rtb_Divide1_h4) || rtIsNaN(rtb_Divide1_h4)) {
    rtb_Divide1_h4 = u0;
  }

  x = Gen2_ref_maximum_f(Gen2_ref_DWork->x_map, inst);
  if ((!(x <= rtb_Divide1_h4)) && (!rtIsNaN(rtb_Divide1_h4))) {
    x = rtb_Divide1_h4;
  }

  k = 0;
  if (!(x < Gen2_ref_DWork->x_map[0])) {
    for (i = 0; i < 13; i++) {
      if (x >= Gen2_ref_DWork->x_map[i]) {
        k = i;
      }
    }
  }

  if (k + 1 < 13) {
    if (Gen2_ref_B->BusInput3.SpeedCtrl.bKF_x_dist1_AdaptON &&
        (!rtb_LogicalOperator_hi)) {
      rtb_Switch_n = Gen2_ref_DWork->y_map[k + 1];
      delta_y_tmp_tmp = x - Gen2_ref_DWork->x_map[k];
      u0 = Gen2_ref_DWork->x_map[k + 1];
      delta_y = delta_y_tmp_tmp / (u0 - Gen2_ref_DWork->x_map[k]) *
        (rtb_Switch_n - Gen2_ref_DWork->y_map[k]) + Gen2_ref_DWork->y_map[k];
      delta_y = ((1.0 - (real_T)Gen2_ref_B->TON_j.LogicalOperator3) * delta_y +
                 (real_T)Gen2_ref_B->TON_j.LogicalOperator3 * rtb_Gain1_o) -
        delta_y;
      x = u0 - x;
      rtb_Gain1_o = delta_y_tmp_tmp + x;
      y_map_tmp = rtb_Gain1_o * x;
      y_map_tmp_0 = (delta_y_tmp_tmp * delta_y_tmp_tmp + y_map_tmp) -
        delta_y_tmp_tmp * x;
      Gen2_ref_DWork->y_map[k] += y_map_tmp * delta_y / y_map_tmp_0;
      Gen2_ref_DWork->y_map[k + 1] = rtb_Gain1_o * delta_y_tmp_tmp * delta_y /
        y_map_tmp_0 + rtb_Switch_n;
    }
  } else if (Gen2_ref_B->BusInput3.SpeedCtrl.bKF_x_dist1_AdaptON &&
             (!rtb_LogicalOperator_hi)) {
    Gen2_ref_DWork->y_map[12] = (1.0 - (real_T)
      Gen2_ref_B->TON_j.LogicalOperator3) * Gen2_ref_DWork->y_map[12] + (real_T)
      Gen2_ref_B->TON_j.LogicalOperator3 * rtb_Gain1_o;
  }
```
